FUNCTION_BLOCK FB_ITC_Conveyor IMPLEMENTS ITF_ITC
(**************************************************************************************
 *  Application     :   BoxControl Framework
 *  Revision date   :   $Date: 2021-04-08 12:45:11 +0200 (tor, 08 apr 2021) $
 *  Author          :   CDC
 *	Purpose			:	ITC - Message Manager.
 *						Represents the interface between the application and the 
 *						communication. Serves as abstract layer to ensure application
 *						independency.
 * ------------------------------------------------------------------------------------
 *  © Swisslog AG
 *  Swisslog is not liable for any usage of this source code that is not agreed 
 *  on between Swisslog and the other party. The mandatory legal liability remains 
 *  unaffected.
 * ------------------------------------------------------------------------------------
 *  Revision History: 
 *
 *  VERSION DATE         INITIALS     DESCRIPTION
 *  0.0     DD.MM.YYYY   (name)       (explain customized modifications)
 *
 **************************************************************************************)
VAR_INPUT
	Config			: ST_CFG_ITC_ManagerConv; // Config
END_VAR

VAR
	Init			: BOOL; // Initialized
	fbDebugMsg		: FB_DebugMsg; // Debug instance
	DebugMsg		: T_MAXSTRING; // Debug msg
	Idx				: INT; // Index for general usage 
	eMsgType		: E_ITC_MsgTypeConv; // Message type conveyor
	Position		: ST_PositionIdent;
	SDI				: ST_ITC_SDI; // SDI
	GVR				: ST_ITC_GVR; // GVR
	ISR				: ST_ITC_ISR; // ISR
	TTC				: ST_ITC_TTC; // TTC
	TDR				: ST_ITC_TDR; // TDR
	FCQ				: ST_ITC_FCQ; // FCQ
	FSR				: ST_ITC_FSR; // FSR
	FSR_Empty		: ST_ITC_FSR; // FSR empty
	SCR				: ST_ITC_SCR; // SCR
	SSR				: ST_ITC_SSR; // SSR
	SSR_Empty		: ST_ITC_SSR; // SSR empty
	GCR				: ST_ITC_GCR; // GCR
	GSR				: ST_ITC_GSR; // GSR
	GSR_Empty		: ST_ITC_GSR; // GSR empty
	ECR				: ST_ITC_ECR; // ECR
	ESR				: ST_ITC_ESR; // ESR
	ESR_Empty		: ST_ITC_ESR; // ESR empty
	FCR				: ST_ITC_FCR; // FCR
	MCR				: ST_ITC_MCR; // MCR
	MCR_Empty		: ST_ITC_MCR; // MCR empty
	SIR				: ST_ITC_SIR; // SIR
	TUR				: ST_ITC_TUR; // TUR
	GDR				: ST_ITC_GDR; // GDR
	GDR_Empty		: ST_ITC_GDR; // GDR empty
	DAR				: ST_ITC_DAR; // DAR
	DAR_Empty		: ST_ITC_DAR; // DAR empty
	Data			: ST_ITC_GeneralData; // General data
	RAC				: ST_ITC_RAC; // RAC
	RDR				: ST_ITC_RDR; // RDR
END_VAR

VAR PERSISTENT
	Settings			: ST_CFG_ITC_ManagerConv; // Active configuration
END_VAR

(**************************************************************************************************************
   Body never called!
***************************************************************************************************************)
;

{attribute 'object_name' := 'M_AddData'}
METHOD M_AddData : BOOL
(**************************************************************************************
 * 	Application		:	BoxControl Framework
 *	Revision		:	$Revision: 474929 $
 *	Revision date	:	$Date: 2021-04-08 12:45:11 +0200 (tor, 08 apr 2021) $
 *	Last changed by	:	$Author: b7gessa $
 *	URL				:	$URL: http://almscdc.swisslog.com/repo/SWPD/Development/BoxControlFramework/20_Release/tags/R1.12.0/01_Software/BCF/BCF/JumpStart/20_Product/10_BCF/11_Conv/11_Com/11_ITC/FB_ITC_Conveyor.TcPOU $
 *
 *	Purpose			:	Add data to the system
 *
 * ------------------------------------------------------------------------------------
 *	Copyright Swisslog [IP AG], Switzerland. All rights reserved.
 * 
 * ------------------------------------------------------------------------------------
 *	
 * 	Revision History: 
 *
 * 	VERSION			DATE			INITIALS			DESCRIPTION
 *	0.1				01.01.2001		swl					Example
 *
 **************************************************************************************)
VAR_INPUT
	meChannelSrc	: E_MFCS_Channel;
	mMsgType		: INT;
	mpData			: PVOID;
	mLen			: UDINT;
END_VAR

M_AddData := FALSE;
// Translate type to enumeration
eMsgType := mMsgType;

// Go to corresponding type
CASE eMsgType OF
	(****************************************************
	  No Message type
	*****************************************************)	
	E_ITC_MsgTypeConv.NO_MESSAGE_TYPE:
		;
	
	(****************************************************
	  Visualization information request
	*****************************************************)	
	E_ITC_MsgTypeConv.VISUALIZATION_INFORMATION_REQUEST:
		// Process
		M_AddData := M_ProcessVIQ(
						meChannelSrc := meChannelSrc,
						mpVIQ := mpData,
						mLen := mLen);
		
	(****************************************************
	  Digital input request
	*****************************************************)	
	E_ITC_MsgTypeConv.DIGITAL_INPUT_REQUEST:
		// Process
		M_AddData := M_ProcessDIQ(
						meChannelSrc := meChannelSrc);
		
	(****************************************************
	  Element control request
	*****************************************************)
	E_ITC_MsgTypeConv.ELEMENT_CONTROL_REQUEST:
		// Process
		M_AddData := M_ProcessECQ(
						meChannelSrc := meChannelSrc,
						mpECQ		 := mpData,
						mLen 		 := mLen);
	
	(****************************************************
	  Element status request
	*****************************************************)		
	E_ITC_MsgTypeConv.ELEMENT_STATUS_REQUEST:
		// Process
		M_AddData := M_ProcessESQ(
						meChannelSrc := meChannelSrc,
						mpESQ		 := mpData,
						mLen 	     := mLen);
		
	(****************************************************
	  Function control request
	*****************************************************)	
	E_ITC_MsgTypeConv.FUNCTION_CONTROL_REQUEST:
		// Process
		M_AddData := M_ProcessFCQ(
						meChannelSrc := meChannelSrc,
						mpFCQ		 := mpData,
						mLen 		 := mLen);
		
	(****************************************************
	  Function status request
	*****************************************************)	
	E_ITC_MsgTypeConv.FUNCTION_STATUS_REQUEST:
		// Process
		M_AddData := M_ProcessFSQ(
						meChannelSrc := meChannelSrc,
						mpFSQ		 := mpData,
						mLen 		 := mLen);
						
	(****************************************************
	  Group control request
	*****************************************************)				
	E_ITC_MsgTypeConv.GROUP_CONTROL_REQUEST:
		// Process
		M_AddData := M_ProcessGCQ(
						meChannelSrc := meChannelSrc,
						mpGCQ		 := mpData,
						mLen 		 := mLen);

	(****************************************************
	  Group status request
	*****************************************************)	
	E_ITC_MsgTypeConv.GROUP_STATUS_REQUEST:
		// Process
		M_AddData := M_ProcessGSQ(
						meChannelSrc := meChannelSrc,
						mpGSQ		 := mpData,
						mLen 		 := mLen);
		
	(****************************************************
	  Global variable request
	*****************************************************)	
	E_ITC_MsgTypeConv.GLOBAL_VARIABLE_REQUEST:
		// Process
		M_AddData := M_ProcessGVQ(
						meChannelSrc := meChannelSrc,
						mpGVQ := mpData,
						mLen := mLen);
						
	(****************************************************
	  IRQ request
	*****************************************************)	
	E_ITC_MsgTypeConv.I_O_STATUS_REQUEST:
		// Process
		M_AddData := M_ProcessIRQ(
						meChannelSrc := meChannelSrc,
						mpIRQ		 := mpData,
						mLen 	     := mLen);
		
	(****************************************************
	  Manual control request
	*****************************************************)					
	E_ITC_MsgTypeConv.MANUAL_CONTROL_REQUEST:
		// Process
		M_AddData := M_ProcessMCQ(
						meChannelSrc := meChannelSrc,
						mpMCQ		 := mpData,
						mLen 		 := mLen);
		
	(****************************************************
	  Robot action assignement
	*****************************************************)					
	E_ITC_MsgTypeConv.ROBOT_ACTION_ASSIGNMENT:
		// Process
		M_AddData := M_ProcessRAA(
						meChannelSrc := meChannelSrc,
						mpRAA		 := mpData,
						mLen 		 := mLen);		
				
	(****************************************************
	  Robot delete request
	*****************************************************)					
	E_ITC_MsgTypeConv.ROBOT_DELETE_REQUEST:
		// Process
		M_AddData := M_ProcessRDQ(
						meChannelSrc := meChannelSrc,
						mpRDQ		 := mpData,
						mLen 		 := mLen);	
			
	(****************************************************
	  Subsystem control request
	*****************************************************)				
	E_ITC_MsgTypeConv.SUBSYSTEM_CONTROL_REQUEST:
		// Process
		M_AddData := M_ProcessSCQ(
						meChannelSrc := meChannelSrc,
						mpSCQ		 := mpData,
						mLen 		 := mLen);
		
	(****************************************************
	  Set digital output
	*****************************************************)				
	E_ITC_MsgTypeConv.SET_DIGITAL_OUTPUT:
		// Process
		M_AddData := M_ProcessSDO(
						meChannelSrc := meChannelSrc,
						mpSDO		 := mpData,
						mLen 		 := mLen);
		
	(****************************************************
	  Scanner information request
	*****************************************************)				
	E_ITC_MsgTypeConv.SCANNER_INFORMATION_REQUEST:
		// Process
		M_AddData := M_ProcessSIQ(
						meChannelSrc := meChannelSrc,
						mpSIQ		 := mpData,
						mLen 		 := mLen);
		
	(****************************************************
	  Subsystem status request
	*****************************************************)			
	E_ITC_MsgTypeConv.SUBSYSTEM_STATUS_REQUEST:
		// Process
		M_AddData := M_ProcessSSQ(
						meChannelSrc := meChannelSrc,
						mpSSQ		 := mpData,
						mLen 		 := mLen);
		
	(****************************************************
	  Task delete request
	*****************************************************)			
	E_ITC_MsgTypeConv.TASK_DELETE_REQUEST:
		// Process
		M_AddData := M_ProcessTDQ(
						meChannelSrc := meChannelSrc,
						mpTDQ		 := mpData,
						mLen 		 := mLen);
		
	(****************************************************
	  Transport task assignment
	*****************************************************)	
	E_ITC_MsgTypeConv.TRANSPORT_TASK_ASSIGNMENT:
		// Process
		M_AddData := M_ProcessTTA(
						meChannelSrc := meChannelSrc,
						mpTTA		 := mpData,
						mLen 		 := mLen);
		
	(****************************************************
	  Transport unit request
	*****************************************************)	
	E_ITC_MsgTypeConv.TRANSPORT_UNIT_REQUEST:
		// Process
		M_AddData := M_ProcessTUQ(
						meChannelSrc := meChannelSrc,
						mpTUQ		 := mpData,
						mLen 	     := mLen);

	(****************************************************
	  Add TU data index into function
	*****************************************************)	
	E_ITC_MsgTypeConv.ADD_TU_DATA:
		// Process
		M_AddData := M_AddTUData(
						meChannelSrc := meChannelSrc,
						mpAddTU_Data		 := mpData);					


						
	(****************************************************
		Data Aquisition Request 
	*****************************************************)	
	E_ITC_MsgTypeConv.DATA_ACQUISITION_REQUEST:
		// Process
		M_AddData := M_ProcessDAQ(
						meChannelSrc := meChannelSrc,
						mpDAQ		 := mpData,
						mLen 	     := mLen);
	(****************************************************
		Gathered Data  Request 
	*****************************************************)	
	E_ITC_MsgTypeConv.GATHERED_DATA_REQUEST:
		// Process
		M_AddData := M_ProcessGDQ(
						meChannelSrc := meChannelSrc,
						mpGDQ		 := mpData,
						mLen 	     := mLen);				
ELSE
	// Unknown type
	DebugMsg := 'Unknown message type received';
	fbDebugMsg.M_SendErrorMsg(mMessage := DebugMsg);		
END_CASE
END_METHOD

METHOD PROTECTED M_AddTUData : BOOL

(**************************************************************************************
 * 	Application		:	BoxControl Framework
 *	Revision		:	$Revision: 474929 $
 *	Revision date	:	$Date: 2021-04-08 12:45:11 +0200 (tor, 08 apr 2021) $
 *	Last changed by	:	$Author: b7gessa $
 *	URL				:	$URL: http://almscdc.swisslog.com/repo/SWPD/Development/BoxControlFramework/20_Release/tags/R1.12.0/01_Software/BCF/BCF/JumpStart/20_Product/10_BCF/11_Conv/11_Com/11_ITC/FB_ITC_Conveyor.TcPOU $
 *
 *	Purpose			:	Process a received Digital Input Request telegram.
 *
 * ------------------------------------------------------------------------------------
 *	Copyright Swisslog [IP AG], Switzerland. All rights reserved.
 * 
 * ------------------------------------------------------------------------------------
 *	
 * 	Revision History: 
 *
 * 	VERSION			DATE			INITIALS			DESCRIPTION
 *	0.1				01.01.2001		swl					Example
 *
 **************************************************************************************)
VAR_INPUT
	meChannelSrc		: E_MFCS_Channel; // Source communicaton channel
	mpAddTU_Data		: POINTER TO ST_ITC_ADD_TU_DATA; // Pointer to SCQ
END_VAR
Data.Init := TRUE;
Data.TU_DataIndex := mpAddTU_Data^.TU_DataIndex;
Data.ZoneNumber := mpAddTU_Data^.ZoneNumber;
Data.Position := '';

// Forward to position
M_AddTUData := M_ProcessToFunction(
	meFunctionNumber	:= mpAddTU_Data^.eFunctionNumber, 
	meChannelSrc		:= meChannelSrc, 
	mMsgType			:= E_ITC_MsgTypeConv.ADD_TU_DATA,
	mpData				:= ADR(Data), 
	mLen				:= SIZEOF(Data));
END_METHOD

{attribute 'object_name' := 'M_CallITC_Service'}
METHOD M_CallITC_Service : BOOL
VAR
	mIdx : INT;
END_VAR
(**************************************************************************************************************
 	Initialization
***************************************************************************************************************)
M_Init(FALSE);

(**************************************************************************************************************
  Monitor SDI Signals
***************************************************************************************************************)
FOR mIdx := 1 TO Settings.SDI_Limit DO
	// SDI signal is enabled 
	IF SDISignalNumber[mIdx].Enabled THEN
		// SDI signal changed state 
		IF SDISignalNumber[mIdx].State <> SDISignalNumber[mIdx].LastState THEN
			// Send SDI
			F_ITC_SendSDI(
				eChannelSrc		:= 0, 
				SignalNumber	:= mIdx, 
				SignalState		:= SDISignalNumber[mIdx].State, 
				eReturnCode		:= E_ErrorConv.NO_ERROR_CODE);
				
			// Update state
			SDISignalNumber[mIdx].LastState := SDISignalNumber[mIdx].State;
		END_IF
	END_IF
END_FOR
END_METHOD

METHOD M_Init : BOOL
(**************************************************************************************
 * 	Application		:	BoxControl Framework
 *	Revision		:	$Revision: 474929 $
 *	Revision date	:	$Date: 2021-04-08 12:45:11 +0200 (tor, 08 apr 2021) $
 *	Last changed by	:	$Author: b7gessa $
 *	URL				:	$URL: http://almscdc.swisslog.com/repo/SWPD/Development/BoxControlFramework/20_Release/tags/R1.12.0/01_Software/BCF/BCF/JumpStart/20_Product/10_BCF/11_Conv/11_Com/11_ITC/FB_ITC_Conveyor.TcPOU $
 *
 *	Purpose			:	Initialize.
 *
 * ------------------------------------------------------------------------------------
 *	Copyright Swisslog [IP AG], Switzerland. All rights reserved.
 * 
 * ------------------------------------------------------------------------------------
 *	
 * 	Revision History: 
 *
 * 	VERSION			DATE			INITIALS			DESCRIPTION
 *	0.1				01.01.2001		swl					Example
 *
 **************************************************************************************)
VAR_INPUT
	mInit		: BOOL; // Force init
END_VAR
// If instance is not initialized or init is forced
IF mInit OR NOT Init THEN
	// Update configuration
	Settings := Config;
	
	// Send log message
    fbDebugMsg.M_SendInfoMsg('Initialization done');
		
	// Init done
    Init := TRUE;
END_IF
END_METHOD

METHOD PRIVATE M_ProcessDAQ : BOOL
(**************************************************************************************
 * 	Application		:	BoxControl Framework
 *	Revision		:	$Revision: 474929 $
 *	Revision date	:	$Date: 2021-04-08 12:45:11 +0200 (tor, 08 apr 2021) $
 *	Last changed by	:	$Author: b7gessa $
 *	URL				:	$URL: http://almscdc.swisslog.com/repo/SWPD/Development/BoxControlFramework/20_Release/tags/R1.12.0/01_Software/BCF/BCF/JumpStart/20_Product/10_BCF/11_Conv/11_Com/11_ITC/FB_ITC_Conveyor.TcPOU $
 *
 *	Purpose			:	Process a received Data Aquisition telegram.
 *
 * ------------------------------------------------------------------------------------
 *	Copyright Swisslog [IP AG], Switzerland. All rights reserved.
 * 
 * ------------------------------------------------------------------------------------
 *	
 * 	Revision History: 
 *
 * 	VERSION			DATE			INITIALS			DESCRIPTION
 *	0.1				01.01.2001		swl					Example
 *
 **************************************************************************************)
VAR_INPUT
	meChannelSrc		: E_MFCS_Channel; // Source communicaton channel
	mpDAQ				: POINTER TO ST_ITC_DAQ; // Pointer to DAQ
	mLen				: UDINT; // Data length
END_VAR
VAR
	meFunctionPosition		: ST_PositionIdent; // Position
	meGroupNumber			: E_GroupNumber; // Group
	meElementNumber			: E_ElementNumber;//Element Number
	meSubsystem				: BOOL;	//Subsystem
	mReturnCode				: E_ErrorConv; // Error code

END_VAR
// Initialize
M_ProcessDAQ:= TRUE;

//Check where position is
meFunctionPosition := F_SearchFunctionPosition(Position := mpDAQ^.Position);
meElementNumber    := F_SearchElementPosition(ElementName := mpDAQ^.Position);
meGroupNumber      := F_SearchGroupNumber(GroupName := mpDAQ^.Position);
meSubsystem 	   := F_EqualSisNames(Name1 := SubsystemRegistry.SubSystemName,
									Name2 := mpDAQ^.Position);

// Check if Function Number is valid
IF meFunctionPosition.eFunctionNumber >F_BEGIN_FUNCTION AND
	meFunctionPosition.eFunctionNumber <F_END_FUNCTION THEN 
    // Forward to Function
	M_ProcessDAQ := M_ProcessToFunction(
						meFunctionNumber:= 	meFunctionPosition.eFunctionNumber, // Position
						meChannelSrc	:= meChannelSrc, 
						mpData			:= mpDAQ, 
						mMsgType		:= E_ITC_MsgTypeConv.DATA_ACQUISITION_REQUEST,
						mLen			:= mLen);
// Check if DAQ was sent to an Element	
ELSIF meElementNumber > E_ElementNumber.E_BEGIN_ELEMENT AND 
      meElementNumber < E_ElementNumber.E_END_ELEMENT AND
      meFunctionPosition.eFunctionNumber = F_BEGIN_FUNCTION AND
      meFunctionPosition.ZoneNumber = 0 THEN 
		// Forward to element
		M_ProcessDAQ := M_ProcessToElement(
						meElementNumber	:= meElementNumber, 
						meChannelSrc	:= meChannelSrc, 
						mpData			:= mpDAQ, 
						mMsgType		:= E_ITC_MsgTypeConv.DATA_ACQUISITION_REQUEST,
						mLen			:= mLen);
// Check if DAQ was sent to a Group					
ELSIF  meGroupNumber > E_GroupNumber.G_BEGIN_GROUP AND 
   		meGroupNumber < E_GroupNumber.G_END_GROUP   AND
		meElementNumber 					= E_BEGIN_ELEMENT AND 
      	meFunctionPosition.eFunctionNumber 	= F_BEGIN_FUNCTION AND
      	meFunctionPosition.ZoneNumber 		= 0 THEN 	   
		// Forward to Group
		M_ProcessDAQ := M_ProcessToGroup(
							meGroupNumber	:= meGroupNumber, // Groupnumber
							meChannelSrc	:= meChannelSrc, 
							mpData			:= mpDAQ, 
							mMsgType		:= E_ITC_MsgTypeConv.DATA_ACQUISITION_REQUEST,
							mLen			:= mLen);
// Check if DAQ was sent to a SubSystem
ELSIF  meSubsystem AND
	   meGroupNumber = G_BEGIN_GROUP AND
	   meElementNumber = E_BEGIN_ELEMENT AND 
	   meFunctionPosition.eFunctionNumber = F_BEGIN_FUNCTION AND
	   meFunctionPosition.ZoneNumber = 0 THEN 	   		
	// Forward to Subsytem						
	M_ProcessDAQ := M_ProcessToSubsystem(
						meChannelSrc	:= meChannelSrc, 
						mpData			:= mpDAQ, 
						mMsgType		:= E_ITC_MsgTypeConv.DATA_ACQUISITION_REQUEST,
						mLen			:= mLen);					
ELSE
	//Unknown position send DAR with Error Report	
	DAR := DAR_Empty;
	// DAR
	DAR.Position	:= mpDAQ^.Position;
	DAR.eErrorCode	:= E_ErrorConv.ELEMENTNUMBER_UNKNOWN;

	// Reject telegram	
	M_SendData(
		meChannel := meChannelSrc,
		mMsgType  := E_ITC_MsgTypeConv.DATA_ACQUISITION_REPORT,
		mpData    := ADR(DAR),
		mLen	  := SIZEOF(DAR));
		
	// Unknown Position name received
	DebugMsg := CONCAT('DAQ - unknown Position name received: ', mpDAQ^.Position);
	fbDebugMsg.M_SendErrorMsg(mMessage := DebugMsg);
END_IF
END_METHOD

METHOD PROTECTED M_ProcessDIQ : BOOL
(**************************************************************************************
 * 	Application		:	BoxControl Framework
 *	Revision		:	$Revision: 474929 $
 *	Revision date	:	$Date: 2021-04-08 12:45:11 +0200 (tor, 08 apr 2021) $
 *	Last changed by	:	$Author: b7gessa $
 *	URL				:	$URL: http://almscdc.swisslog.com/repo/SWPD/Development/BoxControlFramework/20_Release/tags/R1.12.0/01_Software/BCF/BCF/JumpStart/20_Product/10_BCF/11_Conv/11_Com/11_ITC/FB_ITC_Conveyor.TcPOU $
 *
 *	Purpose			:	Process a received Digital Input Request telegram.
 *
 * ------------------------------------------------------------------------------------
 *	Copyright Swisslog [IP AG], Switzerland. All rights reserved.
 * 
 * ------------------------------------------------------------------------------------
 *	
 * 	Revision History: 
 *
 * 	VERSION			DATE			INITIALS			DESCRIPTION
 *	0.1				01.01.2001		swl					Example
 *
 **************************************************************************************)
VAR_INPUT
	meChannelSrc			: E_MFCS_Channel; // Source communicaton channel
END_VAR
// Compose an SDI telegram for every enabled SDI signal
FOR Idx := 1 TO NUMBER_OF_SDI_SIGNALS DO
	// For all enabled SDI SignalNumbers
	IF SDISignalNumber[Idx].Enabled THEN
		// Collect data
		SDI.SignalNumber := Idx;
		SDI.SignalState  := SDISignalNumber[Idx].State;
		SDI.ReturnCode	 := E_ErrorConv.NO_ERROR_CODE;
	
		M_SendData(
			meChannel := meChannelSrc, 
			mMsgType  := E_ITC_MsgTypeConv.SEND_DIGITAL_INPUT, 
			mpData    := ADR(SDI),
			mLen	  := SIZEOF(SDI));
	END_IF
END_FOR

// Telegram processed
M_ProcessDIQ := TRUE;
END_METHOD

METHOD PROTECTED M_ProcessECQ : BOOL
(**************************************************************************************
 * 	Application		:	BoxControl Framework
 *	Revision		:	$Revision: 474929 $
 *	Revision date	:	$Date: 2021-04-08 12:45:11 +0200 (tor, 08 apr 2021) $
 *	Last changed by	:	$Author: b7gessa $
 *	URL				:	$URL: http://almscdc.swisslog.com/repo/SWPD/Development/BoxControlFramework/20_Release/tags/R1.12.0/01_Software/BCF/BCF/JumpStart/20_Product/10_BCF/11_Conv/11_Com/11_ITC/FB_ITC_Conveyor.TcPOU $
 *
 *	Purpose			:	Process a received Element Control Request 
 *
 * ------------------------------------------------------------------------------------
 *	Copyright Swisslog [IP AG], Switzerland. All rights reserved.
 * 
 * ------------------------------------------------------------------------------------
 *	
 * 	Revision History: 
 *
 * 	VERSION			DATE			INITIALS			DESCRIPTION
 *	0.1				01.01.2001		swl					Example
 *
 **************************************************************************************)
VAR_INPUT
	meChannelSrc		: E_MFCS_Channel; // Source communicaton channel
	mpECQ				: POINTER TO ST_ITC_ECQ; // Pointer to ECQ
	mLen				: UDINT; // Data length
END_VAR

VAR
	meElementNumber		: E_ElementNumber; // Element number
END_VAR
// Initialize
M_ProcessECQ := TRUE;

// Try getting enum
meElementNumber := F_SearchElementPosition(ElementName := mpECQ^.Position);

// Check if ElementNumber is valid
IF meElementNumber > E_ElementNumber.E_BEGIN_ELEMENT AND 
   meElementNumber < E_ElementNumber.E_END_ELEMENT THEN
			
	// Forward to element
	M_ProcessECQ := M_ProcessToElement(
						meElementNumber	:= meElementNumber, 
						meChannelSrc	:= meChannelSrc, 
						mMsgType		:= E_ITC_MsgTypeConv.ELEMENT_CONTROL_REQUEST,
						mpData			:= mpECQ, 
						mLen			:= mLen);
						
ELSE
	// Unknown Position name received
	// ECR
	ECR.Position	:= mpECQ^.Position;
	ECR.Code		:= mpECQ^.Code;
	ECR.Variable	:= mpECQ^.Variable;
	ECR.ReturnCode	:= E_ErrorConv.ELEMENTNUMBER_UNKNOWN;

	// Reject telegram	
	M_SendData(
		meChannel := meChannelSrc,
		mMsgType  := E_ITC_MsgTypeConv.ELEMENT_CONTROL_REPLY,
		mpData    := ADR(ECR),
		mLen	  := SIZEOF(ECR));
		
	// Unknown Position name received
	DebugMsg := CONCAT('ECQ - unknown Position name received: ', mpECQ^.Position);
	fbDebugMsg.M_SendErrorMsg(mMessage := DebugMsg);
END_IF
END_METHOD

METHOD PROTECTED M_ProcessESQ : BOOL
(**************************************************************************************
 * 	Application		:	BoxControl Framework
 *	Revision		:	$Revision: 474929 $
 *	Revision date	:	$Date: 2021-04-08 12:45:11 +0200 (tor, 08 apr 2021) $
 *	Last changed by	:	$Author: b7gessa $
 *	URL				:	$URL: http://almscdc.swisslog.com/repo/SWPD/Development/BoxControlFramework/20_Release/tags/R1.12.0/01_Software/BCF/BCF/JumpStart/20_Product/10_BCF/11_Conv/11_Com/11_ITC/FB_ITC_Conveyor.TcPOU $
 *
 *	Purpose			:	Process a received Element Status Request telegram.
 *
 * ------------------------------------------------------------------------------------
 *	Copyright Swisslog [IP AG], Switzerland. All rights reserved.
 * 
 * ------------------------------------------------------------------------------------
 *	
 * 	Revision History: 
 *
 * 	VERSION			DATE			INITIALS			DESCRIPTION
 *	0.1				01.01.2001		swl					Example
 *
 **************************************************************************************)
VAR_INPUT
	meChannelSrc		: E_MFCS_Channel; // Source communicaton channel
	mpESQ				: POINTER TO ST_ITC_ESQ; // Pointer to ESQ
	mLen				: UDINT; // Data length
END_VAR

VAR
	meElementNumber		: E_ElementNumber; // Element number
END_VAR
// Initialize
M_ProcessESQ := TRUE;

// Try getting enum
meElementNumber := F_SearchElementPosition(ElementName := mpESQ^.Position);

// Check if ElementNumber is valid
IF meElementNumber > E_ElementNumber.E_BEGIN_ELEMENT AND 
   meElementNumber < E_ElementNumber.E_END_ELEMENT THEN			
	
	// Forward to element
	M_ProcessESQ := M_ProcessToElement(
						meElementNumber	:= meElementNumber, 
						meChannelSrc	:= meChannelSrc, 
						mMsgType		:= E_ITC_MsgTypeConv.ELEMENT_STATUS_REQUEST,
						mpData			:= mpESQ, 
						mLen			:= mLen);
						
// Check if ESQ was sent to a SubSystem
ELSIF F_EqualSisNames(Name1 := SubsystemRegistry.SubSystemName,
                      Name2 := mpESQ^.Position) THEN
									
	// Do for each ElementNumber
	FOR meElementNumber := E_ElementNumber.E_BEGIN_ELEMENT + 1 TO E_ElementNumber.E_END_Element - 1 DO
		// Forward
		M_ProcessToElement(
			meElementNumber	:= meElementNumber, 
			meChannelSrc	:= meChannelSrc, 
			mMsgType		:= E_ITC_MsgTypeConv.ELEMENT_STATUS_REQUEST,
			mpData			:= mpESQ, 
			mLen			:= mLen);
	END_FOR
ELSE
	ESR := ESR_Empty;
	// Unknown Position name received
	// ESR
	ESR.Position	:= mpESQ^.Position;
	ESR.ReturnCode	:= E_ErrorConv.ELEMENTNUMBER_UNKNOWN;

	// Reject telegram	
	M_SendData(
		meChannel := meChannelSrc,
		mMsgType  := E_ITC_MsgTypeConv.ELEMENT_STATUS_REPORT,
		mpData    := ADR(ESR),
		mLen	  := SIZEOF(ESR));
		
	// Unknown Position name received
	DebugMsg := CONCAT('ESQ - unknown Position name received: ', mpESQ^.Position);
	fbDebugMsg.M_SendErrorMsg(mMessage := DebugMsg);
END_IF
END_METHOD

METHOD PROTECTED M_ProcessFCQ : BOOL
(**************************************************************************************
 * 	Application		:	BoxControl Framework
 *	Revision		:	$Revision: 474929 $
 *	Revision date	:	$Date: 2021-04-08 12:45:11 +0200 (tor, 08 apr 2021) $
 *	Last changed by	:	$Author: b7gessa $
 *	URL				:	$URL: http://almscdc.swisslog.com/repo/SWPD/Development/BoxControlFramework/20_Release/tags/R1.12.0/01_Software/BCF/BCF/JumpStart/20_Product/10_BCF/11_Conv/11_Com/11_ITC/FB_ITC_Conveyor.TcPOU $
 *
 *	Purpose			:	Process a received Function Control Request.
 *
 * ------------------------------------------------------------------------------------
 *	Copyright Swisslog [IP AG], Switzerland. All rights reserved.
 * 
 * ------------------------------------------------------------------------------------
 *	
 * 	Revision History: 
 *
 * 	VERSION			DATE			INITIALS			DESCRIPTION
 *	0.1				01.01.2001		swl					Example
 *
 **************************************************************************************)
VAR_INPUT
	meChannelSrc		: E_MFCS_Channel; // Source communicaton channel
	mpFCQ				: POINTER TO ST_ITC_FCQ; // Pointer to FCQ
	mLen				: UDINT; // Data length
END_VAR

VAR
	mMsgPosition		: ST_PositionIdent; // Function position
	mrefObject			: REFERENCE TO FB_BaseObject; // Reference
END_VAR
// Initialize
M_ProcessFCQ := TRUE;

// Get position from message
mMsgPosition := F_SearchFunctionPosition(Position := mpFCQ^.Position);

// If a valid function was found with a valid zone
IF 	mMsgPosition.eFunctionNumber > E_FunctionNumber.F_BEGIN_FUNCTION AND 
	mMsgPosition.eFunctionNumber < E_FunctionNumber.F_END_FUNCTION AND 
	mMsgPosition.ZoneNumber >= 0 AND mMsgPosition.ZoneNumber <= NUMBER_OF_ZONES_PER_FUNCTION THEN
	
	// Forward to element
	M_ProcessFCQ := M_ProcessToFunction(
						meFunctionNumber	:= mMsgPosition.eFunctionNumber, 
						meChannelSrc		:= meChannelSrc, 
						mMsgType			:= E_ITC_MsgTypeConv.FUNCTION_CONTROL_REQUEST,
						mpData				:= mpFCQ, 
						mLen				:= mLen);
						
ELSE
	// FCR
	FCR.Position	:= mpFCQ^.Position;
	FCR.Code		:= mpFCQ^.Code;
	FCR.Variable	:= mpFCQ^.Variable;
	FCR.ReturnCode	:= E_ErrorConv.FUNCTIONNUMBER_UNKNOWN;

	// Reject telegram	
	M_SendData(
		meChannel := meChannelSrc,
		mMsgType  := E_ITC_MsgTypeConv.FUNCTION_CONTROL_REPLY,
		mpData    := ADR(FCR),
        mLen	  := SIZEOF(FCR));
		
	// Unknown Position name received 
	DebugMsg := CONCAT('FCQ, Unknown Position received: ', mpFCQ^.Position);
	fbDebugMsg.M_SendErrorMsg(mMessage := DebugMsg); 
END_IF
END_METHOD

METHOD PROTECTED M_ProcessFSQ : BOOL
(**************************************************************************************
 * 	Application		:	BoxControl Framework
 *	Revision		:	$Revision: 474929 $
 *	Revision date	:	$Date: 2021-04-08 12:45:11 +0200 (tor, 08 apr 2021) $
 *	Last changed by	:	$Author: b7gessa $
 *	URL				:	$URL: http://almscdc.swisslog.com/repo/SWPD/Development/BoxControlFramework/20_Release/tags/R1.12.0/01_Software/BCF/BCF/JumpStart/20_Product/10_BCF/11_Conv/11_Com/11_ITC/FB_ITC_Conveyor.TcPOU $
 *
 *	Purpose			:	Process a received position Status Request telegram.
 *
 * ------------------------------------------------------------------------------------
 *	Copyright Swisslog [IP AG], Switzerland. All rights reserved.
 * 
 * ------------------------------------------------------------------------------------
 *	
 * 	Revision History: 
 *
 * 	VERSION			DATE			INITIALS			DESCRIPTION
 *	0.1				01.01.2001		swl					Example
 *
 **************************************************************************************)
VAR_INPUT
	meChannelSrc		: E_MFCS_Channel; // Source communicaton channel
	mpFSQ				: POINTER TO ST_ITC_FSQ; // Pointer to FSQ
	mLen				: UDINT; // Data length
END_VAR

VAR
	mMsgPosition		: ST_PositionIdent; // Function position
	mrefObject			: REFERENCE TO FB_BaseObject; // Reference
END_VAR
// Initialize
M_ProcessFSQ := TRUE;

// Get position from message
mMsgPosition := F_SearchFunctionPosition(Position := mpFSQ^.Position);

// If a valid function was found with a valid zone
IF 	mMsgPosition.eFunctionNumber > E_FunctionNumber.F_BEGIN_FUNCTION AND 
	mMsgPosition.eFunctionNumber < E_FunctionNumber.F_END_FUNCTION AND 
	mMsgPosition.ZoneNumber >= 0 AND mMsgPosition.ZoneNumber <= NUMBER_OF_ZONES_PER_FUNCTION THEN

	// Forward to element
	M_ProcessFSQ := M_ProcessToFunction(
						meFunctionNumber	:= mMsgPosition.eFunctionNumber, 
						meChannelSrc		:= meChannelSrc, 
						mMsgType			:= E_ITC_MsgTypeConv.FUNCTION_STATUS_REQUEST,
						mpData				:= mpFSQ,
						mLen				:= mLen);

ELSE
	
	FSR := FSR_Empty;
	
	// FSR
	FSR.Position	:= mpFSQ^.Position;
	FSR.eReturnCode	:= E_ErrorConv.FUNCTIONNUMBER_UNKNOWN;

	// Reject telegram	
	M_SendData(
		meChannel := meChannelSrc,
		mMsgType  := E_ITC_MsgTypeConv.FUNCTION_STATUS_REPORT,
		mpData    := ADR(FSR),
		mLen	  := SIZEOF(FSR));
		
	// Unknown Position name received 
	DebugMsg := CONCAT('FSQ, Unknown Position received: ', mpFSQ^.Position);
	fbDebugMsg.M_SendErrorMsg(mMessage := DebugMsg); 
END_IF
END_METHOD

METHOD PROTECTED M_ProcessGCQ : BOOL
(**************************************************************************************
 * 	Application		:	BoxControl Framework
 *	Revision		:	$Revision: 474929 $
 *	Revision date	:	$Date: 2021-04-08 12:45:11 +0200 (tor, 08 apr 2021) $
 *	Last changed by	:	$Author: b7gessa $
 *	URL				:	$URL: http://almscdc.swisslog.com/repo/SWPD/Development/BoxControlFramework/20_Release/tags/R1.12.0/01_Software/BCF/BCF/JumpStart/20_Product/10_BCF/11_Conv/11_Com/11_ITC/FB_ITC_Conveyor.TcPOU $
 *
 *	Purpose			:	Process a received Group Control Request telegram.
 *
 * ------------------------------------------------------------------------------------
 *	Copyright Swisslog [IP AG], Switzerland. All rights reserved.
 * 
 * ------------------------------------------------------------------------------------
 *	
 * 	Revision History: 
 *
 * 	VERSION			DATE			INITIALS			DESCRIPTION
 *	0.1				01.01.2001		swl					Example
 *
 **************************************************************************************)
VAR_INPUT
	meChannelSrc		: E_MFCS_Channel; // Source communicaton channel
	mpGCQ				: POINTER TO ST_ITC_GCQ; // Pointer to GCQ
	mLen				: UDINT; // Data length
END_VAR

VAR
	meGroupNumber		: E_GroupNumber; // group number
END_VAR
// Initialize 
M_ProcessGCQ := TRUE;

// Find GropuNumber of telegram
meGroupNumber := F_SearchGroupNumber(GroupName := mpGCQ^.Position);
			
// Group number valid
IF meGroupNumber > E_GroupNumber.G_BEGIN_GROUP AND 
   meGroupNumber < E_GroupNumber.G_END_GROUP THEN	
				
	// Forward to group
	M_ProcessGCQ := M_ProcessToGroup(
						meGroupNumber	:= meGroupNumber, 
						meChannelSrc	:= meChannelSrc, 
						mMsgType		:= E_ITC_MsgTypeConv.GROUP_CONTROL_REQUEST,
						mpData			:= mpGCQ, 
						mLen			:= mLen);
				
// Check if GCQ was sent to a SubSystem
ELSIF F_EqualSisNames(Name1 := SubsystemRegistry.SubSystemName,
                      Name2 := mpGCQ^.Position) THEN
			
	// Do for each GroupNumber
	FOR meGroupNumber := E_GroupNumber.G_BEGIN_GROUP + 1 TO E_GroupNumber.G_END_GROUP - 1 DO
		// Check if group is a switching group
		IF GroupRegistry[meGroupNumber].eGroupType = E_GroupType.SG THEN
			M_ProcessToGroup(
				meGroupNumber	:= meGroupNumber, 
				meChannelSrc	:= meChannelSrc, 
				mMsgType		:= E_ITC_MsgTypeConv.GROUP_CONTROL_REQUEST,
				mpData			:= mpGCQ, 
				mLen 			:= mLen);
		END_IF
	END_FOR
ELSE
	
	// GCR
	GCR.GroupName	:= mpGCQ^.Position;
	GCR.Code		:= mpGCQ^.Code;
	GCR.Variable	:= mpGCQ^.Variable;
	GCR.ReturnCode	:= E_ErrorConv.GROUPNUMBER_UNKNOWN;

	// Reject telegram	
	M_SendData(
		meChannel := meChannelSrc,
		mMsgType  := E_ITC_MsgTypeConv.GROUP_CONTROL_REPLY,
		mpData    := ADR(GCR),
		mLen	  := SIZEOF(GCR));

	// Unknown Group name received
	DebugMsg := CONCAT('GCQ, unknown Group name received: ', mpGCQ^.Position);
	fbDebugMsg.M_SendErrorMsg(mMessage := DebugMsg);
END_IF
END_METHOD

METHOD PROTECTED M_ProcessGDQ : BOOL
(**************************************************************************************
 * 	Application		:	BoxControl Framework
 *	Revision		:	$Revision: 474929 $
 *	Revision date	:	$Date: 2021-04-08 12:45:11 +0200 (tor, 08 apr 2021) $
 *	Last changed by	:	$Author: b7gessa $
 *	URL				:	$URL: http://almscdc.swisslog.com/repo/SWPD/Development/BoxControlFramework/20_Release/tags/R1.12.0/01_Software/BCF/BCF/JumpStart/20_Product/10_BCF/11_Conv/11_Com/11_ITC/FB_ITC_Conveyor.TcPOU $
 *
 *	Purpose			:	Process a received Gathered Data Request telegram.
 *
 * ------------------------------------------------------------------------------------
 *	Copyright Swisslog [IP AG], Switzerland. All rights reserved.
 * 
 * ------------------------------------------------------------------------------------
 *	
 * 	Revision History: 
 *
 * 	VERSION			DATE			INITIALS			DESCRIPTION
 *	0.1				01.01.2001		swl					Example
 *
 **************************************************************************************)
VAR_INPUT
	meChannelSrc		: E_MFCS_Channel; // Source communicaton channel
	mpGDQ				: POINTER TO ST_ITC_GDQ; // Pointer to GDQ
	mLen				: UDINT; // Data length
END_VAR
VAR
	meFunctionPosition				: ST_PositionIdent; // Position
	meGroupNumber					: E_GroupNumber; // Group
	meElementNumber					: E_ElementNumber;//Element Number
	meSubsystem						: BOOL;	
	mReturnCode						: E_ErrorConv; // Error code
END_VAR
// Initialize
M_ProcessGDQ:= TRUE;

//Search Position
meFunctionPosition := F_SearchFunctionPosition(Position := mpGDQ^.Position);
meElementNumber    := F_SearchElementPosition(ElementName := mpGDQ^.Position);
meGroupNumber      := F_SearchGroupNumber(GroupName := mpGDQ^.Position);
meSubsystem 	   := F_EqualSisNames(Name1 := SubsystemRegistry.SubSystemName,
														        Name2 := mpGDQ^.Position);

// Check if Function is Target for Telgram 
IF meFunctionPosition.eFunctionNumber >F_BEGIN_FUNCTION AND
	meFunctionPosition.eFunctionNumber <F_END_FUNCTION THEN 
    // Forward to Function
	M_ProcessGDQ := M_ProcessToFunction(
						meFunctionNumber:= 	meFunctionPosition.eFunctionNumber, // Position
						meChannelSrc	:= meChannelSrc, 
						mpData			:= mpGDQ, 
						mMsgType		:= E_ITC_MsgTypeConv.GATHERED_DATA_REQUEST,
						mLen			:= mLen);
// Check if Element is Target for Telgram 
ELSIF meElementNumber > E_ElementNumber.E_BEGIN_ELEMENT AND 
      meElementNumber < E_ElementNumber.E_END_ELEMENT AND
      meFunctionPosition.eFunctionNumber = F_BEGIN_FUNCTION AND
      meFunctionPosition.ZoneNumber = 0 THEN 
	// Forward to element
	M_ProcessGDQ := M_ProcessToElement(
						meElementNumber	:= meElementNumber, 
						meChannelSrc	:= meChannelSrc, 
						mpData			:= mpGDQ, 
						mMsgType		:= E_ITC_MsgTypeConv.GATHERED_DATA_REQUEST,
						mLen			:= mLen);

// Check if Group is Target for Telgram 				
ELSIF  	meGroupNumber > E_GroupNumber.G_BEGIN_GROUP AND 
   		meGroupNumber < E_GroupNumber.G_END_GROUP   AND
		meElementNumber 					= E_BEGIN_ELEMENT AND 
      	meFunctionPosition.eFunctionNumber 	= F_BEGIN_FUNCTION AND
      	meFunctionPosition.ZoneNumber 		= 0 THEN 	   
			
		// Forward to Group
		M_ProcessGDQ := M_ProcessToGroup(
											meGroupNumber	:= meGroupNumber, // Groupnumber
											meChannelSrc	:= meChannelSrc, 
											mpData			:= mpGDQ, 
											mMsgType		:= E_ITC_MsgTypeConv.GATHERED_DATA_REQUEST,
											mLen			:= mLen);
	 
		
// Check if Subystem Target for Telgram 
ELSIF  meSubsystem AND
	   meGroupNumber = G_BEGIN_GROUP AND
	   meElementNumber = E_BEGIN_ELEMENT AND 
	   meFunctionPosition.eFunctionNumber = F_BEGIN_FUNCTION AND
	   meFunctionPosition.ZoneNumber = 0 THEN 	   	
		// Forward to Subsytem			
		M_ProcessGDQ := M_ProcessToSubsystem(
							meChannelSrc	:= meChannelSrc, 
							mpData			:= mpGDQ, 
							mMsgType		:= E_ITC_MsgTypeConv.GATHERED_DATA_REQUEST,
							mLen			:= mLen);
						
		
					
ELSE
	//Unknown position send DAR with Error Report	
	GDR := GDR_Empty;
	
	// DAR
	GDR.Position	:= mpGDQ^.Position;
	GDR.eReturnCode	:= E_ErrorConv.CONFIGURATION_ERROR;

	// Reject telegram	
	M_SendData(
		meChannel := meChannelSrc,
		mMsgType  := E_ITC_MsgTypeConv.GATHERED_DATA_REQUEST,
		mpData    := ADR(GDR),
		mLen	  := mLen );
		
	// Unknown Position name received
	DebugMsg := CONCAT('GDQ - unknown Position name received: ', mpGDQ^.Position);
	fbDebugMsg.M_SendErrorMsg(mMessage := DebugMsg);
END_IF
END_METHOD

METHOD PROTECTED M_ProcessGSQ : BOOL
(**************************************************************************************
 * 	Application		:	BoxControl Framework
 *	Revision		:	$Revision: 474929 $
 *	Revision date	:	$Date: 2021-04-08 12:45:11 +0200 (tor, 08 apr 2021) $
 *	Last changed by	:	$Author: b7gessa $
 *	URL				:	$URL: http://almscdc.swisslog.com/repo/SWPD/Development/BoxControlFramework/20_Release/tags/R1.12.0/01_Software/BCF/BCF/JumpStart/20_Product/10_BCF/11_Conv/11_Com/11_ITC/FB_ITC_Conveyor.TcPOU $
 *
 *	Purpose			:	Process a received Group Status Request telegram.
 *
 * ------------------------------------------------------------------------------------
 *	Copyright Swisslog [IP AG], Switzerland. All rights reserved.
 * 
 * ------------------------------------------------------------------------------------
 *	
 * 	Revision History: 
 *
 * 	VERSION			DATE			INITIALS			DESCRIPTION
 *	0.1				01.01.2001		swl					Example
 *
 **************************************************************************************)
VAR_INPUT
	meChannelSrc		: E_MFCS_Channel; // Source communicaton channel
	mpGSQ				: POINTER TO ST_ITC_GSQ; // Pointer to GSQ
	mLen				: UDINT; // Data length
END_VAR

VAR
	meGroupNumber		: E_GroupNumber; // group number
END_VAR
// Initialize
M_ProcessGSQ := TRUE;

// Find GropuNumber of telegram
meGroupNumber := F_SearchGroupNumber(GroupName := mpGSQ^.Position);
			
// Request was for a group
// Group number valid
IF meGroupNumber > E_GroupNumber.G_BEGIN_GROUP AND 
   meGroupNumber < E_GroupNumber.G_END_GROUP THEN	
						
	// Forward to group
	M_ProcessGSQ := M_ProcessToGroup(
						meGroupNumber	:= meGroupNumber, 
						meChannelSrc	:= meChannelSrc, 
						mMsgType		:= E_ITC_MsgTypeConv.GROUP_STATUS_REQUEST,
						mpData			:= mpGSQ,
						mLen			:= mLen);
					
// Check if GCQ was sent to a SubSystem
ELSIF F_EqualSisNames(Name1 := SubsystemRegistry.SubSystemName,
                      Name2 := mpGSQ^.Position) THEN
			
	// Do for each GroupNumber
	FOR meGroupNumber := E_GroupNumber.G_BEGIN_GROUP + 1 TO E_GroupNumber.G_END_GROUP - 1 DO
		
		M_ProcessToGroup(
			meGroupNumber	:= meGroupNumber, 
			meChannelSrc	:= meChannelSrc, 
			mMsgType		:= E_ITC_MsgTypeConv.GROUP_STATUS_REQUEST,
			mpData			:= mpGSQ, 
			mLen			:= mLen);
	END_FOR
	
ELSE
	GSR := GSR_Empty;
	
	// GSR
	GSR.GroupName	:= mpGSQ^.Position;
	GSR.eReturnCode	:= E_ErrorConv.GROUPNUMBER_UNKNOWN;

	// Reject telegram	
	M_SendData(
		meChannel := meChannelSrc,
		mMsgType  := E_ITC_MsgTypeConv.GROUP_STATUS_REPORT,
		mpData    := ADR(GSR),
		mLen	  := SIZEOF(GSR));
		
	// Unknown Group name received
	DebugMsg := CONCAT('GSQ, unknown Group name received: ', mpGSQ^.Position);
	fbDebugMsg.M_SendErrorMsg(mMessage := DebugMsg);
END_IF
END_METHOD

METHOD PROTECTED M_ProcessGVQ : BOOL
(**************************************************************************************
 * 	Application		:	BoxControl Framework
 *	Revision		:	$Revision: 474929 $
 *	Revision date	:	$Date: 2021-04-08 12:45:11 +0200 (tor, 08 apr 2021) $
 *	Last changed by	:	$Author: b7gessa $
 *	URL				:	$URL: http://almscdc.swisslog.com/repo/SWPD/Development/BoxControlFramework/20_Release/tags/R1.12.0/01_Software/BCF/BCF/JumpStart/20_Product/10_BCF/11_Conv/11_Com/11_ITC/FB_ITC_Conveyor.TcPOU $
 *
 *	Purpose			:	Process a received Global Variable Request telegram.
 *
 * ------------------------------------------------------------------------------------
 *	Copyright Swisslog [IP AG], Switzerland. All rights reserved.
 * 
 * ------------------------------------------------------------------------------------
 *	
 * 	Revision History: 
 *
 * 	VERSION			DATE			INITIALS			DESCRIPTION
 *	0.1				01.01.2001		swl					Example
 *
 **************************************************************************************)
VAR_INPUT
	meChannelSrc		: E_MFCS_Channel; // Source communicaton channel
	mpGVQ				: POINTER TO ST_ITC_GVQ; // Pointer to GVQ
	mLen				: UDINT; // Data length
END_VAR

VAR
	mIdx				: INT; // Iterator
	mError				: BOOL; // Error during processing
	mVar				: ARRAY[0..9] OF DINT; // Temporary variables
END_VAR
// Initialize
M_ProcessGVQ := TRUE;

// Initialize
mError := FALSE;

// Check borders
IF mpGVQ^.Number > GVR_Table.NUMBER_OF_GVR_SIGNALS OR
   mpGVQ^.Number < 1  OR
   mpGVQ^.Quantity < 1 OR
   mpGVQ^.Quantity > 10 THEN
	// Set error
	mError := TRUE;
END_IF

// If no error is active
IF NOT mError THEN
	// If perform action is selected
	IF mpGVQ^.Code = 1 OR mpGVQ^.Code = 2 THEN
		// Map values
		mVar[0] := mpGVQ^.Variable[0];
		mVar[1] := mpGVQ^.Variable[1];
		mVar[2] := mpGVQ^.Variable[2];
		mVar[3] := mpGVQ^.Variable[3];
		mVar[4] := mpGVQ^.Variable[4];
		mVar[5] := mpGVQ^.Variable[5];
		mVar[6] := mpGVQ^.Variable[6];
		mVar[7] := mpGVQ^.Variable[7];
		mVar[8] := mpGVQ^.Variable[8];
		mVar[9] := mpGVQ^.Variable[9];
	   
		// Go trough quantity
		FOR mIdx := 0 TO mpGVQ^.Quantity - 1 DO
			// Set values
			GlobalVariable[mpGVQ^.Number, mIdx] := mVar[mIdx];
		END_FOR
	END_IF
	
	// If report state is selected
	IF mpGVQ^.Code = 0 OR mpGVQ^.Code = 2 THEN
		GVR.Number := mpGVQ^.Number;
		GVR.Quantity := mpGVQ^.Quantity;
		
		// Go trough quantity
		FOR mIdx := 0 TO 9 DO
			// Set values
			GVR.Variable[mIdx] := 0;
		END_FOR
		
		FOR mIdx := 0 TO mpGVQ^.Quantity - 1 DO
			// Set values
			GVR.Variable[mIdx] := GlobalVariable[mpGVQ^.Number, mIdx];
		END_FOR

		GVR.ReturnCode := E_ErrorConv.NO_ERROR_CODE;
	
		M_SendData(
			meChannel := meChannelSrc, 
			mMsgType  := E_ITC_MsgTypeConv.GLOBAL_VARIABLE_REPORT, 
			mpData    := ADR(GVR),
			mLen	  := SIZEOF(GVR));
	END_IF
ELSE
	GVR.Number := mpGVQ^.Number;
	GVR.Quantity := mpGVQ^.Quantity;
	GVR.Variable[0] :=0;
	GVR.Variable[1] := 0;
	GVR.Variable[2] := 0;
	GVR.Variable[3] := 0;
	GVR.Variable[4] := 0;
	GVR.Variable[5] := 0;
	GVR.Variable[6] := 0;
	GVR.Variable[7] := 0;
	GVR.Variable[8] := 0;
	GVR.Variable[9] := 0;
	GVR.ReturnCode := E_ErrorConv.WRONG_VALUE;

	M_SendData(
		meChannel := meChannelSrc, 
		mMsgType  := E_ITC_MsgTypeConv.GLOBAL_VARIABLE_REPORT, 
		mpData    := ADR(GVR),
		mLen	  := SIZEOF(GVR));
END_IF
END_METHOD

METHOD PROTECTED M_ProcessIRQ : BOOL
(**************************************************************************************
 * 	Application		:	BoxControl Framework
 *	Revision		:	$Revision: 474929 $
 *	Revision date	:	$Date: 2021-04-08 12:45:11 +0200 (tor, 08 apr 2021) $
 *	Last changed by	:	$Author: b7gessa $
 *	URL				:	$URL: http://almscdc.swisslog.com/repo/SWPD/Development/BoxControlFramework/20_Release/tags/R1.12.0/01_Software/BCF/BCF/JumpStart/20_Product/10_BCF/11_Conv/11_Com/11_ITC/FB_ITC_Conveyor.TcPOU $
 *
 *	Purpose			:	Process a received I/O Status Request telegram.
 *
 * ------------------------------------------------------------------------------------
 *	Copyright Swisslog [IP AG], Switzerland. All rights reserved.
 * 
 * ------------------------------------------------------------------------------------
 *	
 * 	Revision History: 
 *
 * 	VERSION			DATE			INITIALS			DESCRIPTION
 *	0.1				01.01.2001		swl					Example
 *
 **************************************************************************************)
VAR_INPUT
	meChannelSrc		: E_MFCS_Channel; // Source communicaton channel
	mpIRQ				: POINTER TO ST_ITC_IRQ; // Pointer to IRQ
	mLen				: UDINT; // Data length
END_VAR


VAR
	mInformation		: STRING(NUMBER_OF_ISR_DATA_LENGTH); // Internal information
	mSignalNumber		: INT; // SignalNumber
	mIdx				: INT; // Internal cunter
	mByte				: BYTE; // Internal Byte
END_VAR
// Initialize
M_ProcessIRQ := TRUE;

// Init String
mInformation := '';

// Get the signal data for each block of 4 requested
// an mDataLength of 01 actually means get 4 bits
FOR mIdx := 1 TO mpIRQ^.DataLength BY 1 DO
	
	// Calculate base signal number
	mSignalNumber  := (((mIdx - 1) * 4) + mpIRQ^.StartSignalNumber);
	// Init Byte
	mByte := 0;

	// Check if we will remain in range of the ISR Signal numbers
	IF (mSignalNumber + 4) <= NUMBER_OF_ISR_SIGNALS THEN
		// Get the signal state for this group of 4 and put them in the correct bits
		mByte.0 := ISR_SignalType[mpIRQ^.SignalType].SignalNumber[mSignalNumber];
		mByte.1 := ISR_SignalType[mpIRQ^.SignalType].SignalNumber[mSignalNumber + 1];
		mByte.2 := ISR_SignalType[mpIRQ^.SignalType].SignalNumber[mSignalNumber + 2];
		mByte.3 := ISR_SignalType[mpIRQ^.SignalType].SignalNumber[mSignalNumber + 3];
	END_IF

	// Convert the resultant tByte to a value between '0' and 'F'
	fbFormatString (sFormat := '%X', arg1 := F_BYTE(mByte));

	// Add the ASCII result for this block of 4 bits to the ISR.Information string
	mInformation := CONCAT(mInformation, fbFormatString.sOut);
END_FOR

(* Information string should always be 99 chars long
   therefore pad mInformation with trailing zeros. *)
FOR mIdx := LEN(mInformation) TO NUMBER_OF_ISR_DATA_LENGTH DO
	mInformation := CONCAT(mInformation, '0');
END_FOR

// Collect data
ISR.DataLength := mpIRQ^.DataLength;
ISR.Information := mInformation;
ISR.SignalType := mpIRQ^.SignalType;
ISR.StartSignalNumber := mpIRQ^.StartSignalNumber;
ISR.ReturnCode := E_ErrorConv.NO_ERROR_CODE;

M_SendData(
	meChannel := meChannelSrc, 
	mMsgType  := E_ITC_MsgTypeConv.I_O_STATUS_REPORT, 
	mpData    := ADR(ISR),
	mLen	  := SIZEOF(ISR));
END_METHOD

METHOD PROTECTED M_ProcessMCQ : BOOL
(**************************************************************************************
 * 	Application		:	BoxControl Framework
 *	Revision		:	$Revision: 474929 $
 *	Revision date	:	$Date: 2021-04-08 12:45:11 +0200 (tor, 08 apr 2021) $
 *	Last changed by	:	$Author: b7gessa $
 *	URL				:	$URL: http://almscdc.swisslog.com/repo/SWPD/Development/BoxControlFramework/20_Release/tags/R1.12.0/01_Software/BCF/BCF/JumpStart/20_Product/10_BCF/11_Conv/11_Com/11_ITC/FB_ITC_Conveyor.TcPOU $
 *
 *	Purpose			:	Process a received Manual Control Request telegram.
 *
 * ------------------------------------------------------------------------------------
 *	Copyright Swisslog [IP AG], Switzerland. All rights reserved.
 * 
 * ------------------------------------------------------------------------------------
 *	
 * 	Revision History: 
 *
 * 	VERSION			DATE			INITIALS			DESCRIPTION
 *	0.1				01.01.2001		swl					Example
 *
 **************************************************************************************)
VAR_INPUT
	meChannelSrc		: E_MFCS_Channel; // Source communicaton channel
	mpMCQ				: POINTER TO ST_ITC_MCQ; // Pointer to MCQ
	mLen				: UDINT; // Data length
END_VAR

VAR
	meElementNumber			: E_ElementNumber; // PositionNumber
	mFunction				: ST_PositionIdent; // Function
END_VAR

// Initialize
M_ProcessMCQ := TRUE;

// Get element number
meElementNumber := F_SearchElementPosition(ElementName := mpMCQ^.Position);

// Get function
mFunction := F_SearchFunctionPosition(Position := mpMCQ^.Position);

// Valid ElementNumber was found
IF meElementNumber > E_ElementNumber.E_BEGIN_ELEMENT AND meElementNumber < E_ElementNumber.E_END_ELEMENT THEN

	// Forward to element
	M_ProcessMCQ := M_ProcessToElement(
						meElementNumber	:= meElementNumber, 
						meChannelSrc	:= meChannelSrc, 
						mMsgType		:= E_ITC_MsgTypeConv.MANUAL_CONTROL_REQUEST,
						mpData			:= mpMCQ,
						mLen			:= mLen);		
		
// Valid FunctionNumber was found
ELSIF mFunction.eFunctionNumber > E_FunctionNumber.F_BEGIN_FUNCTION AND 
      mFunction.eFunctionNumber < E_FunctionNumber.F_END_FUNCTION THEN
	
	// Forward to function
	M_ProcessMCQ := M_ProcessToFunction(
						meFunctionNumber	:= mFunction.eFunctionNumber, 
						meChannelSrc		:= meChannelSrc, 
						mMsgType			:= E_ITC_MsgTypeConv.MANUAL_CONTROL_REQUEST,
						mpData				:= mpMCQ,
						mLen				:= mLen);
	
ELSE
	// Unknown name received
	MCR := MCR_Empty;	

	MCR.Position := mpMCQ^.Position;
	MCR.Mode := E_PositionMode.UNKNOWN_MODE;
	MCR.Code := mpMCQ^.Code;
	MCR.eReturnCode := E_ErrorConv.WRONG_VALUE;

	// Reject telegram	
	M_SendData(
		meChannel := meChannelSrc,
		mMsgType  := E_ITC_MsgTypeConv.MANUAL_CONTROL_REPORT,
		mpData    := ADR(MCR),
		mLen	  := SIZEOF(MCR));
		
	// Unknown name received
	DebugMsg := CONCAT('MCQ, unknown Position name received: ', mpMCQ^.Position);
	fbDebugMsg.M_SendErrorMsg(mMessage := DebugMsg);
END_IF
END_METHOD

METHOD PROTECTED M_ProcessRAA : BOOL
(**************************************************************************************
 * 	Application		:	BoxControl Framework
 *	Revision		:	$Revision: 474929 $
 *	Revision date	:	$Date: 2021-04-08 12:45:11 +0200 (tor, 08 apr 2021) $
 *	Last changed by	:	$Author: b7gessa $
 *	URL				:	$URL: http://almscdc.swisslog.com/repo/SWPD/Development/BoxControlFramework/20_Release/tags/R1.12.0/01_Software/BCF/BCF/JumpStart/20_Product/10_BCF/11_Conv/11_Com/11_ITC/FB_ITC_Conveyor.TcPOU $
 *
 *	Purpose			:	Process a received Transport Task Assignment telegram for a robot.
 *
 * ------------------------------------------------------------------------------------
 *	Copyright Swisslog [IP AG], Switzerland. All rights reserved.
 * 
 * ------------------------------------------------------------------------------------
 *	
 * 	Revision History: 
 *
 * VERSION DATE         INITIALS     DESCRIPTION
 * 0.0     DD.MM.YYYY   (name)       (explain customized modifications)
 *
 **************************************************************************************)

//***********************************************************************************************************
VAR_INPUT
  meChannelSrc          : E_MFCS_Channel         := 0;     // Source communicaton channel
  mpRAA                 : POINTER TO ST_ITC_RAA  := 0;     // Pointer to RAA
  mLen                  : UDINT                  := 0;     // Data length
END_VAR

//***********************************************************************************************************
VAR
  eFunctionNumber       : E_FunctionNumber       := 0;
  eElementNumber        : E_ElementNumber        := 0;
  eGroupNumber          : E_GroupNumber          := 0;
  //-------------------------------------------------------------------------------------
  Subsystem             : BOOL                   := FALSE;
END_VAR

// parse and find requested position
eFunctionNumber:= F_FindFunction  (Name:= mpRAA^.Position);
eElementNumber := F_FindElement   (Name:= mpRAA^.Position);
eGroupNumber   := F_FindGroup     (Name:= mpRAA^.Position);
Subsystem      := F_CheckSubsystem(Name:= mpRAA^.Position);

// to function ?
IF eFunctionNumber <> E_FunctionNumber.F_BEGIN_FUNCTION THEN
	M_ProcessRAA:= M_ProcessToFunction(	meFunctionNumber:= eFunctionNumber, 
										meChannelSrc    := meChannelSrc, 
										mMsgType        := E_ITC_MsgTypeConv.ROBOT_ACTION_ASSIGNMENT,
										mpData          := mpRAA, 
										mLen            := mLen);
	// forwarding successful -> no debug message necessary here


// to element ?
ELSIF eElementNumber <> E_ElementNumber.E_BEGIN_ELEMENT THEN
	M_ProcessRAA:= M_ProcessToElement(	meElementNumber:= eElementNumber,
										meChannelSrc   := meChannelSrc, 
										mMsgType       := E_ITC_MsgTypeConv.ROBOT_ACTION_ASSIGNMENT,
										mpData         := mpRAA, 
										mLen           := mLen);
	// forwarding successful -> no debug message necessary here


// to group ?
ELSIF eGroupNumber <> E_GroupNumber.G_BEGIN_GROUP THEN
	M_ProcessRAA:= M_ProcessToGroup(meGroupNumber:= eGroupNumber,
									meChannelSrc := meChannelSrc, 
									mMsgType     := E_ITC_MsgTypeConv.ROBOT_ACTION_ASSIGNMENT,
									mpData       := mpRAA, 
									mLen         := mLen);
	// forwarding successful -> no debug message necessary here


// to subsystem ?
ELSIF Subsystem THEN
	M_ProcessRAA:= M_ProcessToSubsystem(meChannelSrc:= meChannelSrc, 
										mMsgType    := E_ITC_MsgTypeConv.ROBOT_ACTION_ASSIGNMENT,
										mpData      := mpRAA, 
										mLen        := mLen);
	// forwarding successful -> no debug message necessary here


//* unknown position -> fire error telegram
ELSE
  // reject telegram
	RAC.Position        := mpRAA^.Position;
	RAC.CommandDataIndex:= mpRAA^.CommandDataIndex;
	RAC.GroupID         := mpRAA^.GroupID;
	RAC.AssignmentID    := mpRAA^.AssignmentID;
	RAC.eReturnCode     := E_ErrorConv.FUNCTIONNUMBER_UNKNOWN;
	M_SendData(	meChannel:= meChannelSrc, 
				mMsgType := E_ITC_MsgTypeConv.ROBOT_ACTION_COMPLETE, 
				mpData   := ADR(RAC),
				mLen     := SIZEOF(RAC));	

	// debug message
	// example: '11-000-0000-00-0,  unknown position addressed,  telegram = RAA,  Position = 99-999-9999-99-9,  AssignmentID = 9999999'
	DebugMsg:= '';
	DebugMsg:= CONCAT(DebugMsg, F_AddDividerToSisString(SubsystemRegistry.SubsystemName));
	DebugMsg:= CONCAT(DebugMsg, ', unknown position addressed');
	DebugMsg:= CONCAT(DebugMsg, DebugTextBlocks.TELEGRAM);
	DebugMsg:= CONCAT(DebugMsg, 'RAA');
	DebugMsg:= CONCAT(DebugMsg, DebugTextBlocks.POSITION);
	DebugMsg:= CONCAT(DebugMsg, F_AddDividerToSisString(Name:= mpRAA^.Position)  );
	DebugMsg:= CONCAT(DebugMsg, DebugTextBlocks.ASSIGNMENTID);
	DebugMsg:= CONCAT(DebugMsg, UDINT_TO_STRING(mpRAA^.AssignmentID) );
	fbDebugMsg.M_SendErrorMsg(mMessage := DebugMsg);
	
	// forwarding to here ITC were possible so prevent error message from FB_SIS_MsgManager
	M_ProcessRAA:= TRUE;
END_IF
END_METHOD

METHOD PROTECTED M_ProcessRDQ : BOOL
(**************************************************************************************
 * 	Application		:	BoxControl Framework
 *	Revision		:	$Revision: 474929 $
 *	Revision date	:	$Date: 2021-04-08 12:45:11 +0200 (tor, 08 apr 2021) $
 *	Last changed by	:	$Author: b7gessa $
 *	URL				:	$URL: http://almscdc.swisslog.com/repo/SWPD/Development/BoxControlFramework/20_Release/tags/R1.12.0/01_Software/BCF/BCF/JumpStart/20_Product/10_BCF/11_Conv/11_Com/11_ITC/FB_ITC_Conveyor.TcPOU $
 *
 *	Purpose			:	Robot delete request
 *
 * ------------------------------------------------------------------------------------
 *	Copyright Swisslog [IP AG], Switzerland. All rights reserved.
 * 
 * ------------------------------------------------------------------------------------
 *	
 * 	Revision History: 
 *
 * 	VERSION			DATE			INITIALS			DESCRIPTION
 *	0.1				03.11.2015		Kay Röder			Example
 *
 **************************************************************************************)
VAR_INPUT
	meChannelSrc				: E_MFCS_Channel; // Source communicaton channel
	mpRDQ						: POINTER TO ST_ITC_RDQ; // Pointer to EDQ
	mLen						: UDINT; // Data length
END_VAR

VAR
	mMsgPosition		: ST_PositionIdent; // Function position
	mReturnCode 		: U_ErrorCode;
END_VAR
// Initialize
M_ProcessRDQ := TRUE;
	   
// Get position from message
mMsgPosition := F_SearchFunctionPosition(Position := mpRDQ^.Position);
	
// If a valid function was found with a valid zone
IF 	mMsgPosition.eFunctionNumber > E_FunctionNumber.F_BEGIN_FUNCTION AND 
	mMsgPosition.eFunctionNumber < E_FunctionNumber.F_END_FUNCTION AND 
	mMsgPosition.ZoneNumber >= 0 AND mMsgPosition.ZoneNumber <= NUMBER_OF_ZONES_PER_FUNCTION THEN
	
	// Forward to element
	M_ProcessRDQ := M_ProcessToFunction(
						meFunctionNumber	:= mMsgPosition.eFunctionNumber, 
						meChannelSrc		:= meChannelSrc, 
						mMsgType			:= E_ITC_MsgTypeConv.ROBOT_DELETE_REQUEST,
						mpData				:= mpRDQ, 
						mLen				:= mLen);
				
	DebugMsg := CONCAT('Robot Delete Assignment Request: ', UDINT_TO_STRING(mpRDQ^.AssignmentID));
	fbDebugMsg.M_SendInfoMsg(mMessage := DebugMsg);
 
ELSE
	mReturnCode.Conv := E_ErrorConv.FUNCTIONNUMBER_UNKNOWN; 
	
	// Reject telegram	
	RDR.Position := mpRDQ^.Position;
	RDR.CommandDataIndex := mpRDQ^.CommandDataIndex;
	RDR.GroupID := mpRDQ^.GroupID;
	RDR.AssignmentID := 0;
	RDR.ReturnCode := mReturnCode.Conv;

	M_SendData(
		meChannel := meChannelSrc, 
		mMsgType  := E_ITC_MsgTypeConv.ROBOT_DELETE_REPORT, 
		mpData    := ADR(RDR),
		mLen	  := SIZEOF(RDR));

	DebugMsg := CONCAT('Robot Delete Assignment Request: ', UDINT_TO_STRING(mpRDQ^.AssignmentID));
	DebugMsg := CONCAT(DebugMsg, 'has an invalid ITC config on RowPaQ-PLC-project');
	fbDebugMsg.M_SendErrorMsg(mMessage := DebugMsg);
END_IF
END_METHOD

METHOD PROTECTED M_ProcessSCQ : BOOL
(**************************************************************************************
 * 	Application		:	BoxControl Framework
 *	Revision		:	$Revision: 474929 $
 *	Revision date	:	$Date: 2021-04-08 12:45:11 +0200 (tor, 08 apr 2021) $
 *	Last changed by	:	$Author: b7gessa $
 *	URL				:	$URL: http://almscdc.swisslog.com/repo/SWPD/Development/BoxControlFramework/20_Release/tags/R1.12.0/01_Software/BCF/BCF/JumpStart/20_Product/10_BCF/11_Conv/11_Com/11_ITC/FB_ITC_Conveyor.TcPOU $
 *
 *	Purpose			:	Process a received Subsystem Control Request telegram.
 *
 * ------------------------------------------------------------------------------------
 *	Copyright Swisslog [IP AG], Switzerland. All rights reserved.
 * 
 * ------------------------------------------------------------------------------------
 *	
 * 	Revision History: 
 *
 * 	VERSION			DATE			INITIALS			DESCRIPTION
 *	0.1				01.01.2001		swl					Example
 *
 **************************************************************************************)
VAR_INPUT
	meChannelSrc		: E_MFCS_Channel; // Source communicaton channel
	mpSCQ				: POINTER TO ST_ITC_SCQ; // Pointer to SCQ
	mLen				: UDINT; // Data length
END_VAR
// Initialize 
M_ProcessSCQ := TRUE;

// Check if SubSystem is valid
IF F_EqualSisNames(Name1 := SubsystemRegistry.SubSystemName,
                   Name2 := mpSCQ^.SubsystemName) THEN
		
	// Forward to subsystem
	M_ProcessSCQ := M_ProcessToSubsystem(
						meChannelSrc	:= meChannelSrc, 
						mMsgType		:= E_ITC_MsgTypeConv.SUBSYSTEM_CONTROL_REQUEST,
						mpData			:= mpSCQ,
						mLen			:= mLen);		
ELSE
	// Unknown SubSystem number received
	SCR.SubsystemName	:= mpSCQ^.SubsystemName;
	SCR.Code			:= mpSCQ^.Code;
	SCR.Variable		:= mpSCQ^.Variable;
	SCR.ReturnCode		:= E_ErrorConv.SubsystemNUMBER_UNKNOWN;

	// Reject telegram	
	M_SendData(
		meChannel := meChannelSrc,
		mMsgType  := E_ITC_MsgTypeConv.SUBSYSTEM_CONTROL_REPLY,
		mpData    := ADR(SCR),
		mLen	  := SIZEOF(SCR));

	// Unknown SubSystem number received
	DebugMsg := CONCAT('SCQ, unknown SubSystem name received: ', mpSCQ^.SubsystemName);
	fbDebugMsg.M_SendErrorMsg(mMessage := DebugMsg);
END_IF
END_METHOD

METHOD PROTECTED M_ProcessSDO : BOOL
(**************************************************************************************
 * 	Application		:	BoxControl Framework
 *	Revision		:	$Revision: 474929 $
 *	Revision date	:	$Date: 2021-04-08 12:45:11 +0200 (tor, 08 apr 2021) $
 *	Last changed by	:	$Author: b7gessa $
 *	URL				:	$URL: http://almscdc.swisslog.com/repo/SWPD/Development/BoxControlFramework/20_Release/tags/R1.12.0/01_Software/BCF/BCF/JumpStart/20_Product/10_BCF/11_Conv/11_Com/11_ITC/FB_ITC_Conveyor.TcPOU $
 *
 *	Purpose			:	Process a received Set Digital Output telegram.
 *						Set or Reset the appropriate SDO signal number according 
 *						to the data in the telegram
 *
 * ------------------------------------------------------------------------------------
 *	Copyright Swisslog [IP AG], Switzerland. All rights reserved.
 * 
 * ------------------------------------------------------------------------------------
 *	
 * 	Revision History: 
 *
 * 	VERSION			DATE			INITIALS			DESCRIPTION
 *	0.1				01.01.2001		swl					Example
 *
 **************************************************************************************)
VAR_INPUT
	meChannelSrc		: E_MFCS_Channel; // Source communicaton channel
	mpSDO				: POINTER TO ST_ITC_SDO; // Pointer to SCQ
	mLen				: UDINT; // Data length
END_VAR
// Initialize
M_ProcessSDO := TRUE;

// Range check the SignalNumber
IF mpSDO^.SignalNumber > 0 THEN
	// Set SignalState
	SDOSignalNumber[mpSDO^.SignalNumber] := INT_TO_BOOL(mpSDO^.SignalState);
END_IF
END_METHOD

METHOD PROTECTED M_ProcessSIQ : BOOL
(**************************************************************************************
 * 	Application		:	BoxControl Framework
 *	Revision		:	$Revision: 474929 $
 *	Revision date	:	$Date: 2021-04-08 12:45:11 +0200 (tor, 08 apr 2021) $
 *	Last changed by	:	$Author: b7gessa $
 *	URL				:	$URL: http://almscdc.swisslog.com/repo/SWPD/Development/BoxControlFramework/20_Release/tags/R1.12.0/01_Software/BCF/BCF/JumpStart/20_Product/10_BCF/11_Conv/11_Com/11_ITC/FB_ITC_Conveyor.TcPOU $
 *
 *	Purpose			:	Process a received Scanner Information Request telegram.
 *
 * ------------------------------------------------------------------------------------
 *	Copyright Swisslog [IP AG], Switzerland. All rights reserved.
 * 
 * ------------------------------------------------------------------------------------
 *	
 * 	Revision History: 
 *
 * 	VERSION			DATE			INITIALS			DESCRIPTION
 *	0.1				01.01.2001		swl					Example
 *
 **************************************************************************************)
VAR_INPUT
	meChannelSrc		: E_MFCS_Channel; // Source communicaton channel
	mpSIQ				: POINTER TO ST_ITC_SIQ; // Pointer to SIQ
	mLen				: UDINT; // Data length
END_VAR

VAR
	mFunction			: ST_PositionIdent; // Function position
END_VAR
// Initialize
M_ProcessSIQ := TRUE;

//Find element function of telegram
mFunction := F_SearchFunctionPosition(Position := mpSIQ^.Position);

// If function number is valid
IF mFunction.eFunctionNumber > E_FunctionNumber.F_BEGIN_FUNCTION AND 
   mFunction.eFunctionNumber < E_FunctionNumber.F_END_FUNCTION THEN
   
	// Forward to function
	M_ProcessSIQ := M_ProcessToFunction(
						meFunctionNumber	:= mFunction.eFunctionNumber,
						meChannelSrc		:= meChannelSrc, 
						mMsgType			:= E_ITC_MsgTypeConv.SCANNER_INFORMATION_REQUEST,
						mpData				:= mpSIQ, 
						mLen				:= mLen);

ELSE
	// Unknown Position name received
	SIR.Position := mpSIQ^.Position;
	SIR.Code := mpSIQ^.Code;
	SIR.TU_ID := '';
	SIR.Counter1 := 0;
	SIR.Counter2 := 0;
	SIR.Counter3 := 0;
	SIR.Counter4 := 0;
	SIR.Counter5 := 0;
	SIR.eReturnCode := E_ErrorConv.FUNCTIONNUMBER_UNKNOWN;

	// Reject telegram	
	M_SendData(
		meChannel := meChannelSrc,
		mMsgType  := E_ITC_MsgTypeConv.SCANNER_INFORMATION_REPORT,
		mpData    := ADR(SIR),
		mLen	  := SIZEOF(SIR));

	// Unknown Position name received
	DebugMsg := CONCAT('SIQ, unknown Position name received: ', mpSIQ^.Position);
	fbDebugMsg.M_SendErrorMsg(mMessage := DebugMsg);	
END_IF
END_METHOD

METHOD PROTECTED M_ProcessSSQ : BOOL
(**************************************************************************************
 * 	Application		:	BoxControl Framework
 *	Revision		:	$Revision: 474929 $
 *	Revision date	:	$Date: 2021-04-08 12:45:11 +0200 (tor, 08 apr 2021) $
 *	Last changed by	:	$Author: b7gessa $
 *	URL				:	$URL: http://almscdc.swisslog.com/repo/SWPD/Development/BoxControlFramework/20_Release/tags/R1.12.0/01_Software/BCF/BCF/JumpStart/20_Product/10_BCF/11_Conv/11_Com/11_ITC/FB_ITC_Conveyor.TcPOU $
 *
 *	Purpose			:	Process a received Subsystem Status Request telegram.
 *
 * ------------------------------------------------------------------------------------
 *	Copyright Swisslog [IP AG], Switzerland. All rights reserved.
 * 
 * ------------------------------------------------------------------------------------
 *	
 * 	Revision History: 
 *
 * 	VERSION			DATE			INITIALS			DESCRIPTION
 *	0.1				01.01.2001		swl					Example
 *
 **************************************************************************************)
VAR_INPUT
	meChannelSrc		: E_MFCS_Channel; // Source communicaton channel
	mpSSQ				: POINTER TO ST_ITC_SSQ; // Pointer to SCQ
	mLen				: UDINT; // Data length
END_VAR
// Initialize
M_ProcessSSQ := TRUE;

// Check if SubSystem is valid
IF F_EqualSisNames(Name1 := SubsystemRegistry.SubsystemName,
                   Name2 := mpSSQ^.Position) THEN
		
		// Forward to subsystem
		M_ProcessSSQ := M_ProcessToSubsystem(
							meChannelSrc	:= meChannelSrc, 
							mMsgType		:= E_ITC_MsgTypeConv.SUBSYSTEM_STATUS_REQUEST,
							mpData			:= mpSSQ, 
							mLen			:= mLen);	
ELSE
	SSR := SSR_Empty;
	
	// SSR
	SSR.SubsystemName	:= mpSSQ^.Position;
	SSR.eReturnCode	:= E_ErrorConv.SubsystemNUMBER_UNKNOWN;

	// Reject telegram	
	M_SendData(
		meChannel := meChannelSrc,
		mMsgType  := E_ITC_MsgTypeConv.SUBSYSTEM_STATUS_REPORT,
		mpData    := ADR(SSR),
		mLen	  := SIZEOF(SSR));
		
	// Unknown SubSystem number received
	DebugMsg := CONCAT('SSQ, unknown SubSystem name received: ', mpSSQ^.Position);
	fbDebugMsg.M_SendErrorMsg(mMessage := DebugMsg);
END_IF
END_METHOD

METHOD PROTECTED M_ProcessTDQ : BOOL
(**************************************************************************************
 *  Application     :   BoxControl Framework
 *  Revision date   :   $Date: 2021-04-08 12:45:11 +0200 (tor, 08 apr 2021) $
 *  Author          :   CDC
 * ------------------------------------------------------------------------------------
 *  © Swisslog AG
 *  Swisslog is not liable for any usage of this source code that is not agreed 
 *  on between Swisslog and the other party. The mandatory legal liability remains 
 *  unaffected.
 * ------------------------------------------------------------------------------------
 *  Revision History: 
 *
 *  VERSION DATE         INITIALS     DESCRIPTION
 *  0.0     DD.MM.YYYY   (name)       (explain customized modifications)
 *
 **************************************************************************************)
VAR_INPUT
	meChannelSrc			: E_MFCS_Channel; // Source communicaton channel
	mpTDQ					: POINTER TO ST_ITC_TDQ; // Pointer to TDQ
	mLen					: UDINT; // Data length
END_VAR

VAR
	mPosition				: ST_PositionIdent ; // Position
	mReturnCode				: E_ErrorConv; // Return code
	mTU_ID_Present			: BOOL; // TU-ID present
	mTU_DataIndex			: DINT; // TU-data index
	mAssignmentID_Present	: BOOL; // Assignment-ID present
	mAssignmentID_Index		: DINT; // Assignment-ID index
END_VAR
// Init
mReturnCode := E_ErrorConv.NO_ERROR_CODE;
M_ProcessTDQ := TRUE;
mTU_ID_Present := FALSE;
mTU_DataIndex := 0;
mAssignmentID_Present := FALSE;
mAssignmentID_Index := 0;

// Get position from telegram
mPosition := F_SearchFunctionPosition( Position := mpTDQ^.Position);

// Order to delete all TU-data
IF mpTDQ^.Code = 1 THEN
	// Check no function number and unknown TU-ID
	IF mpTDQ^.TU_ID = Conveyor.TU_ID_UNKNOWN AND mPosition.eFunctionNumber = 0 THEN
		// Check all TU-Data for DataSets
		FOR mTU_DataIndex := 1 TO Conveyor.NUMBER_OF_TU_DATA BY 1 DO
			// Check if TU-DataSet is used
			IF TU_DataTable[mTU_DataIndex].DataSet.DataPresent THEN	
				// debug message: '11-001-0095-01-1,  TU_DataIndex deleted,  telegram = TDQ,  TU_DataIndex = 5,  TuID = 000012345,  AssignmentID = 999999999'
				DebugMsg := '';
				DebugMsg := CONCAT(DebugMsg, F_AddDividerToSisString(mpTDQ^.Position));
				DebugMsg := CONCAT(DebugMsg, ',  TU_DataIndex deleted');
				DebugMsg := CONCAT(DebugMsg, DebugTextBlocks.TELEGRAM);
				DebugMsg := CONCAT(DebugMsg, 'TDQ');
				DebugMsg := CONCAT(DebugMsg, F_CreateTU_DataString(TU_DataIndex:= mTU_DataIndex));
				fbDebugMsg.M_SendInfoMsg(DebugMsg);
				// Delete TU-Data
				F_DeleteTU_Data(
					TU_DataIndex 	:= mTU_DataIndex, // TU_DataIndex from zone
					NoTTC 			:= FALSE); // No TTC will be sent
			END_IF
		END_FOR

		TDR.Position := mpTDQ^.Position;
		TDR.TU_ID := mpTDQ^.TU_ID;
		TDR.AssignmentID := mpTDQ^.AssignmentID;
		TDR.MsgSequence := mpTDQ^.MsgSequence;
		TDR.ReturnCode := mReturnCode;
		
		M_SendData(
			meChannel := meChannelSrc, 
			mMsgType  := E_ITC_MsgTypeConv.TASK_DELETE_REPORT, 
			mpData    := ADR(TDR),
			mLen	  := SIZEOF(TDR));
		RETURN;
	ELSE
		// Error: Wrong value
		mReturnCode := E_ErrorConv.WRONG_VALUE;
	END_IF
	
// Specific request for TU-ID or position
ELSE
	// Check if an Assignment-ID is present
	mAssignmentID_Present := mpTDQ^.AssignmentID > 0 AND mpTDQ^.AssignmentID < Conveyor.ASSIGNMENT_ID_UNKNOWN;
	
	// Check if a TU-ID is present
	mTU_ID_Present := mpTDQ^.TU_ID <> F_StuffString('', Conveyor.TU_ID_STRINGLENGTH,'0', FALSE) AND
				      mpTDQ^.TU_ID <> F_StuffString('', Conveyor.TU_ID_STRINGLENGTH,' ', FALSE);
	
	// If a valid position is found
	IF mPosition.eFunctionNumber > E_FunctionNumber.F_BEGIN_FUNCTION AND
	   mPosition.ZoneNumber > 0 THEN
		// Get TU-data from zone
		mTU_DataIndex := F_GetTU_DataIndex(
								eFunctionNumber := mPosition.eFunctionNumber, // PositionNumber
								ZoneNumber := mPosition.ZoneNumber); // ZoneNumber
		// A TU index was found
		IF mTU_DataIndex > 0 THEN
			IF mAssignmentID_Present THEN
				// Compare received Assignment ID with the Assignment ID from the position
				IF TU_DataTable[mTU_DataIndex].AssignmentID <> mpTDQ^.AssignmentID THEN
					// Error: Wrong Assignement-ID
					mReturnCode := E_ErrorConv.ASSIGNMENT_ID_WRONG;
				END_IF
			ELSIF mTU_ID_Present THEN
				// Compare received TU ID with the TU ID from the position
				IF TU_DataTable[mTU_DataIndex].TU_ID.ASCII <> mpTDQ^.TU_ID THEN
					// Error: Wrong TU-ID
					mReturnCode := E_ErrorConv.TU_ID_WRONG;
				END_IF
			ELSE
				// Error: Wrong value
				mReturnCode := E_ErrorConv.ID_WRONG;
			END_IF
		ELSE
			// Error: No TU data set available on position
			mReturnCode := E_ErrorConv.EMPTY_TU_DATA_SET;
		END_IF
		
	// Request to subsystem
	ELSIF mpTDQ^.Position <> F_ReduceToAlphaNumeric(SubsystemRegistry.SubsystemName) THEN
		// Error: Position wrong 
		mReturnCode := E_ErrorConv.FUNCTIONNUMBER_UNKNOWN;
		
	// Telegram without function number
	ELSE
		IF mAssignmentID_Present THEN
			// Search TU-data index based on the Assignement-ID in the TU-data table
			mAssignmentID_Index := F_SearchAssignmentId(mpTDQ^.AssignmentID);
		END_IF
		
		IF mTU_ID_Present THEN
			// Search TU-data index based on the TU-ID in the TU-data table
			mTU_DataIndex := F_SearchTU_ByHashCode(mpTDQ^.TU_ID);
		END_IF			
		
		// If an Assignement-ID index is found
		IF mAssignmentID_Index <> 0 THEN
			// Search position belonging to the Assignement-ID index
			// to report last position
			mPosition := F_SearchPositionOfTU_Index(
								TU_DataIndex := mAssignmentID_Index, // TU_DataIndex from zone
								eStartFunctionNumber := E_FunctionNumber.F_BEGIN_FUNCTION + 1); // Start Zone
		// If a TU-data index is found
		ELSIF mTU_DataIndex <> 0 THEN
			// Search position belonging to the TU-data index
			// to report last position
			mPosition := F_SearchPositionOfTU_Index(
								TU_DataIndex := mTU_DataIndex, // TU_DataIndex from zone
								eStartFunctionNumber := E_FunctionNumber.F_BEGIN_FUNCTION + 1); // Start Zone
		ELSE
			IF mAssignmentID_Present THEN
				// Error: Wrong Assignement-ID
				mReturnCode := E_ErrorConv.ASSIGNMENT_ID_WRONG;
			ELSIF mTU_ID_Present THEN
				// Error: Wrong TU-ID
				mReturnCode := E_ErrorConv.TU_ID_WRONG;
			ELSE
				// Error: No data
				mReturnCode := E_ErrorConv.ID_WRONG;
			END_IF
		END_IF
	END_IF
END_IF

// Send task delete report
IF mPosition.eFunctionNumber <> E_FunctionNumber.F_BEGIN_FUNCTION THEN
	TDR.Position := F_ReduceToAlphaNumeric(FunctionRegistry[mPosition.eFunctionNumber].Zone[mPosition.ZoneNumber].ZoneName);
ELSE
	TDR.Position := mpTDQ^.Position;
END_IF
TDR.TU_ID := mpTDQ^.TU_ID;
TDR.AssignmentID := mpTDQ^.AssignmentID;
TDR.MsgSequence := mpTDQ^.MsgSequence;
TDR.ReturnCode := mReturnCode;

M_SendData(
	meChannel := meChannelSrc, 
	mMsgType  := E_ITC_MsgTypeConv.TASK_DELETE_REPORT, 
	mpData    := ADR(TDR),
	mLen	  := SIZEOF(TDR));

// Still no error so far
IF mReturnCode = 0  THEN
	// TU-data index available
	IF mTU_DataIndex <> 0 THEN
		// debug message: '11-001-0095-01-1,  TU_DataIndex deleted,  telegram = TDQ,  TU_DataIndex = 5,  TuID = 000012345,  AssignmentID = 999999999'
		DebugMsg := '';
		DebugMsg := CONCAT(DebugMsg, F_AddDividerToSisString(mpTDQ^.Position));
		DebugMsg := CONCAT(DebugMsg, ',  TU_DataIndex deleted');
		DebugMsg := CONCAT(DebugMsg, DebugTextBlocks.TELEGRAM);
		DebugMsg := CONCAT(DebugMsg, 'TDQ');
		DebugMsg := CONCAT(DebugMsg, F_CreateTU_DataString(TU_DataIndex:= mTU_DataIndex));
		fbDebugMsg.M_SendInfoMsg(DebugMsg);
		// Delete TU-data in the system
		F_DeleteTU_Data(
			TU_DataIndex 	:= mTU_DataIndex,
			NoTTC 			:= FALSE);
	// Assignement-ID index available
	ELSIF mAssignmentID_Index <> 0 THEN
		// debug message: '11-001-0095-01-1,  TU_DataIndex deleted,  telegram = TDQ,  TU_DataIndex = 5,  TuID = 000012345,  AssignmentID = 999999999'
		DebugMsg := '';
		DebugMsg := CONCAT(DebugMsg, F_AddDividerToSisString(mpTDQ^.Position));
		DebugMsg := CONCAT(DebugMsg, ',  TU_DataIndex deleted');
		DebugMsg := CONCAT(DebugMsg, DebugTextBlocks.TELEGRAM);
		DebugMsg := CONCAT(DebugMsg, 'TDQ');
		DebugMsg := CONCAT(DebugMsg, F_CreateTU_DataString(TU_DataIndex:= mAssignmentID_Index));
		fbDebugMsg.M_SendInfoMsg(DebugMsg);
		// Delete TU-data in the system
		F_DeleteTU_Data(
			TU_DataIndex 	:= mAssignmentID_Index,
			NoTTC 			:= FALSE);
	ELSE		
		DebugMsg := 'TDQ, Process failed - no TU-index available.';
		fbDebugMsg.M_SendErrorMsg(mMessage := DebugMsg);		
	END_IF
END_IF
END_METHOD

METHOD PROTECTED M_ProcessToElement : BOOL
(**************************************************************************************
 * 	Application		:	BoxControl Framework
 *	Revision		:	$Revision: 474929 $
 *	Revision date	:	$Date: 2021-04-08 12:45:11 +0200 (tor, 08 apr 2021) $
 *	Last changed by	:	$Author: b7gessa $
 *	URL				:	$URL: http://almscdc.swisslog.com/repo/SWPD/Development/BoxControlFramework/20_Release/tags/R1.12.0/01_Software/BCF/BCF/JumpStart/20_Product/10_BCF/11_Conv/11_Com/11_ITC/FB_ITC_Conveyor.TcPOU $
 *
 *	Purpose			:	ITC - Process message to element
 *
 * ------------------------------------------------------------------------------------
 *	Copyright Swisslog [IP AG], Switzerland. All rights reserved.
 * 
 * ------------------------------------------------------------------------------------
 *	
 * 	Revision History: 
 *
 * 	VERSION			DATE			INITIALS			DESCRIPTION
 *	0.1				01.01.2001		swl					Example
 *
 **************************************************************************************)
VAR_INPUT
	meElementNumber	: E_ElementNumber;
	meChannelSrc	: E_MFCS_Channel; // Source communicaton channel
	mMsgType			: INT; // msg type
	mpData				: POINTER TO PVOID; // data pointer
	mLen				: UDINT; // Data length
END_VAR

VAR
	mrefObject		: REFERENCE TO FB_BaseObject; // Reference
END_VAR
// Initialize
M_ProcessToElement := TRUE;

// Check if ElementNumber is valid
IF meElementNumber > E_ElementNumber.E_BEGIN_ELEMENT AND 
   meElementNumber < E_ElementNumber.E_END_ELEMENT THEN
	// Set reference
	mrefObject REF= ElementRegistry[meElementNumber].rElement;
	
	// Check if reference is valid
	IF __ISVALIDREF(mrefObject) THEN
			// Forward message to corresponding object
		M_ProcessToElement := mrefObject.M_ITC_ProcessMsg(
								meChannelSrc := meChannelSrc,
								mMsgType	 := mMsgType,
								mpData		 := mpData,
								mLen		 := mLen); 
	END_IF	
END_IF
END_METHOD

METHOD PROTECTED M_ProcessToFunction : BOOL
(**************************************************************************************
 * 	Application		:	BoxControl Framework
 *	Revision		:	$Revision: 474929 $
 *	Revision date	:	$Date: 2021-04-08 12:45:11 +0200 (tor, 08 apr 2021) $
 *	Last changed by	:	$Author: b7gessa $
 *	URL				:	$URL: http://almscdc.swisslog.com/repo/SWPD/Development/BoxControlFramework/20_Release/tags/R1.12.0/01_Software/BCF/BCF/JumpStart/20_Product/10_BCF/11_Conv/11_Com/11_ITC/FB_ITC_Conveyor.TcPOU $
 *
 *	Purpose			:	ITC - Process message to function
 *
 * ------------------------------------------------------------------------------------
 *	Copyright Swisslog [IP AG], Switzerland. All rights reserved.
 * 
 * ------------------------------------------------------------------------------------
 *	
 * 	Revision History: 
 *
 * 	VERSION			DATE			INITIALS			DESCRIPTION
 *	0.1				01.01.2001		swl					Example
 *
 **************************************************************************************)
VAR_INPUT
	meFunctionNumber	: E_FunctionNumber; // Function number
	meChannelSrc		: E_MFCS_Channel; // Source communicaton channel
	mMsgType			: INT; // msg type
	mpData				: POINTER TO PVOID; // data pointer
	mLen				: UDINT; // Data length
END_VAR

VAR
	mrefObject			: REFERENCE TO FB_BaseObject; // Reference
END_VAR
// Initialize
M_ProcessToFunction := TRUE;

// If a valid function was found with a valid zone
IF 	meFunctionNumber > E_FunctionNumber.F_BEGIN_FUNCTION AND 
	meFunctionNumber < E_FunctionNumber.F_END_FUNCTION THEN

	// Set reference 
	mrefObject REF= FunctionRegistry[meFunctionNumber].rFunction;
	
	// Check if reference is valid
	IF __ISVALIDREF(mrefObject) THEN

		// Call M_ITC_AddToBuffer
		M_ProcessToFunction := mrefObject.M_ITC_ProcessMsg(
								meChannelSrc := meChannelSrc, // Number of the source 
								mMsgType	 := mMsgType, // Type of the ITC message
								mpData		 := mpData,
								mLen		 := mLen); // Data pointer of the message	
	END_IF
END_IF
END_METHOD

METHOD PROTECTED M_ProcessToGroup : BOOL
(**************************************************************************************
 * 	Application		:	BoxControl Framework
 *	Revision		:	$Revision: 474929 $
 *	Revision date	:	$Date: 2021-04-08 12:45:11 +0200 (tor, 08 apr 2021) $
 *	Last changed by	:	$Author: b7gessa $
 *	URL				:	$URL: http://almscdc.swisslog.com/repo/SWPD/Development/BoxControlFramework/20_Release/tags/R1.12.0/01_Software/BCF/BCF/JumpStart/20_Product/10_BCF/11_Conv/11_Com/11_ITC/FB_ITC_Conveyor.TcPOU $
 *
 *	Purpose			:	ITC - Process message to group
 *
 * ------------------------------------------------------------------------------------
 *	Copyright Swisslog [IP AG], Switzerland. All rights reserved.
 * 
 * ------------------------------------------------------------------------------------
 *	
 * 	Revision History: 
 *
 * 	VERSION			DATE			INITIALS			DESCRIPTION
 *	0.1				01.01.2001		swl					Example
 *
 **************************************************************************************)
VAR_INPUT
	meGroupNumber		: E_GroupNumber; // Groupnumber
	meChannelSrc		: E_MFCS_Channel; // Source communicaton channel
	mMsgType			: INT; // msg type
	mpData				: POINTER TO PVOID; // data pointer
	mLen				: UDINT; // Data length
END_VAR

VAR
	mrefObject			: REFERENCE TO FB_BaseObject; // Reference
END_VAR
// Initialize
M_ProcessToGroup := TRUE;

// Check if GroupNumber is valid
IF meGroupNumber > E_GroupNumber.G_BEGIN_GROUP AND 
   meGroupNumber < E_GroupNumber.G_END_GROUP THEN
	// Set reference
	mrefObject REF= GroupRegistry[meGroupNumber].rGroup;
	
	// Check if reference is valid
	IF __ISVALIDREF(mrefObject) THEN
		
		// Send ITC-message to a specified group
		M_ProcessToGroup := mrefObject.M_ITC_ProcessMsg(
								meChannelSrc := meChannelSrc,
								mMsgType	 := mMsgType, 
								mpData		 := mpData,
								mLen		 := mLen); 
	END_IF
END_IF
END_METHOD

METHOD PROTECTED M_ProcessToSubsystem : BOOL
(**************************************************************************************
 * 	Application		:	BoxControl Framework
 *	Revision		:	$Revision: 474929 $
 *	Revision date	:	$Date: 2021-04-08 12:45:11 +0200 (tor, 08 apr 2021) $
 *	Last changed by	:	$Author: b7gessa $
 *	URL				:	$URL: http://almscdc.swisslog.com/repo/SWPD/Development/BoxControlFramework/20_Release/tags/R1.12.0/01_Software/BCF/BCF/JumpStart/20_Product/10_BCF/11_Conv/11_Com/11_ITC/FB_ITC_Conveyor.TcPOU $
 *
 *	Purpose			:	ITC - Process message to subsystem
 *
 * ------------------------------------------------------------------------------------
 *	Copyright Swisslog [IP AG], Switzerland. All rights reserved.
 * 
 * ------------------------------------------------------------------------------------
 *	
 * 	Revision History: 
 *
 * 	VERSION			DATE			INITIALS			DESCRIPTION
 *	0.1				01.01.2001		swl					Example
 *
 **************************************************************************************)
VAR_INPUT
	meChannelSrc		: E_MFCS_Channel; // Source communicaton channel
	mMsgType			: INT; // msg type
	mpData				: POINTER TO PVOID; // data pointer
	mLen				: UDINT; // Data length
END_VAR

VAR
	mrefObject			: REFERENCE TO FB_BaseObject; // Reference
END_VAR
// Initialize
M_ProcessToSubsystem := TRUE;

// Set reference 
mrefObject REF= SubsystemRegistry.rSubsystem;

// Check if reference is valid
IF __ISVALIDREF(mrefObject) THEN
	// Call M_ITC_AddToBuffer
	M_ProcessToSubsystem := mrefObject.M_ITC_ProcessMsg(
								meChannelSrc := meChannelSrc,
								mMsgType	 := mMsgType, 
								mpData		 := mpData,	
								mLen		 := mLen);  
END_IF
END_METHOD

METHOD PROTECTED M_ProcessTTA : BOOL
(**************************************************************************************
 * 	Application		:	BoxControl Framework
 *	Revision		:	$Revision: 474929 $
 *	Revision date	:	$Date: 2021-04-08 12:45:11 +0200 (tor, 08 apr 2021) $
 *	Last changed by	:	$Author: b7gessa $
 *	URL				:	$URL: http://almscdc.swisslog.com/repo/SWPD/Development/BoxControlFramework/20_Release/tags/R1.12.0/01_Software/BCF/BCF/JumpStart/20_Product/10_BCF/11_Conv/11_Com/11_ITC/FB_ITC_Conveyor.TcPOU $
 *
 *	Purpose			:	Process a received Transport Task Assignment telegram.
 *
 * ------------------------------------------------------------------------------------
 *	Copyright Swisslog [IP AG], Switzerland. All rights reserved.
 * 
 * ------------------------------------------------------------------------------------
 *	
 * 	Revision History: 
 *
 * VERSION DATE         INITIALS     DESCRIPTION
 * 0.0     DD.MM.YYYY   (name)       (explain customized modifications)
 *
 **************************************************************************************)
VAR_INPUT
	meChannelSrc				: E_MFCS_Channel; // Source communicaton channel
	mpTTA						: POINTER TO ST_ITC_TTA; // Pointer to TTA
	mLen						: UDINT;
END_VAR

VAR
	mOtherPosition				: ST_PositionIdent; // OtherPosition where same Index is used
	mDestinationPosition		: ARRAY[1..NUMBER_OF_DESTINATIONS] OF ST_PositionIdent; // DestinationPosition
	mVirtualDestinationPosition	: ARRAY[1..NUMBER_OF_DESTINATIONS] OF ST_PositionIdent;
	mReturnCode					: E_ErrorConv; // Error code
	mTU_DataIndexPosition		: DINT; // Data Index from PositionNumber
	mTU_DataIndex				: DINT; // Data Index from Data_ID
	mRequestForPosition			: BOOL; // Request for a Position
	mTransportData				: ST_TransportControlData; // Transport data
	mTU_ID_Present				: BOOL; // TU-ID present
	mAssignmentID_Present		: BOOL; // Assignment ID present
	mAssignmentID_Index			: DINT; // Assignment ID index
	mDestIndex					: INT; // Temporary destination index
END_VAR
// Initialize
M_ProcessTTA := TRUE;
mTU_DataIndexPosition := 0;
mRequestForPosition := FALSE;	
mTU_DataIndex := 0;
mAssignmentID_Index := 0;
mAssignmentID_Present := FALSE;
mTU_ID_Present := FALSE;

(**************************************************************************************
Check if request is valid
***************************************************************************************)
// Search position in registry
Position := F_SearchFunctionPosition(Position := mpTTA^.Position);

//Check if a TU-ID is present
mTU_ID_Present := 	mpTTA^.TU_ID <> F_StuffString('', Conveyor.TU_ID_STRINGLENGTH,'0', FALSE)
				AND mpTTA^.TU_ID <> F_StuffString('', Conveyor.TU_ID_STRINGLENGTH,' ', FALSE);

IF mTU_ID_Present THEN
	// Search if the TU-ID already exists
	mTU_DataIndex := F_SearchTU_ByHashCode(mpTTA^.TU_ID);
END_IF	

// Check if an asssignment-ID is present					   
mAssignmentID_Present := mpTTA^.AssignmentID > 0;

IF mAssignmentID_Present THEN
	// Search if the assignment-ID already exists
	mAssignmentID_Index := F_SearchAssignmentId(mpTTA^.AssignmentID);
END_IF


// If the telegram contains no TU-ID and no assignment-ID
IF NOT mTU_ID_Present AND NOT mAssignmentID_Present THEN
	// Error: ID is wrong 
	mReturnCode := E_ErrorConv.ID_WRONG;
	// debug message: '11-000-0000-00-0,  TuID and AssignmentID missing,  telegram = TTA'
	DebugMsg:= '';
	DebugMsg:= CONCAT(DebugMsg, F_AddDividerToSisString(SubsystemRegistry.SubsystemName));
	DebugMsg:= CONCAT(DebugMsg, ',  TuID and AssignmentID missing');
	DebugMsg:= CONCAT(DebugMsg, DebugTextBlocks.TELEGRAM);
	DebugMsg:= CONCAT(DebugMsg, 'TTA');
	fbDebugMsg.M_SendErrorMsg(mMessage := DebugMsg);


// If the request goes to a position
ELSIF Position.eFunctionNumber > E_FunctionNumber.F_BEGIN_FUNCTION AND 
	Position.eFunctionNumber < E_FunctionNumber.F_END_FUNCTION THEN
	// If a valid zone was found
	IF 	Position.ZoneNumber > 0
	AND Position.ZoneNumber <= NUMBER_OF_ZONES_PER_FUNCTION THEN
		// Get transport data
		mTransportData := F_GetTransportControlData(
		eFunctionNumber := Position.eFunctionNumber,
		ZoneNumber		:= Position.ZoneNumber);
		
		(*	Data can only be added if the location is physically occupied.
			State occupied is not working in this place, because on a system
			with enabled MFC, the place gets occupied only with a physical 
			and a logical unit. *)
		IF mTransportData.SensorOccupied THEN
			// Save - Valid request for a position
			mRequestForPosition := TRUE;	

			// Get TU Index of telegram position
			mTU_DataIndexPosition := F_GetTU_DataIndex( 
			eFunctionNumber := Position.eFunctionNumber,
			ZoneNumber 		:= Position.ZoneNumber);
			// If an index is found
			IF mTU_DataIndexPosition > 0 THEN
			(* 
			Adding data is allowed, if
			- TU-ID of desired position is 'unknown' OR
			- Telegram TU-ID is equal to position TU-ID
			
			AND
			- Position consists of an unknown assignment-ID OR
			- Assignment-ID is equal to the requested one		
			
			AND
			- When a requested Index was available, it needs to be equal to position index		
			*)
				IF (TU_DataTable[mTU_DataIndexPosition].TU_ID.ASCII = Conveyor.TU_ID_UNKNOWN OR 
				mpTTA^.TU_ID = TU_DataTable[mTU_DataIndexPosition].TU_ID.ASCII) AND 
				(mpTTA^.AssignmentID = TU_DataTable[mTU_DataIndexPosition].AssignmentID OR
				Conveyor.ASSIGNMENT_ID_UNKNOWN = TU_DataTable[mTU_DataIndexPosition].AssignmentID) AND
				((mpTTA^.TU_DataIndex > 0 AND mpTTA^.TU_DataIndex = mTU_DataIndexPosition) OR (mpTTA^.TU_DataIndex = 0)) THEN 
					// Adding data is allowed by TU-ID
					;
				// Adding not allowed
				ELSE
					// When the assignment-ID was not equal to the already existing or 
					// the assignment-ID on the position was not unknown
					IF TU_DataTable[mTU_DataIndexPosition].AssignmentID <> mpTTA^.AssignmentID AND 
					   TU_DataTable[mTU_DataIndexPosition].AssignmentID <> Conveyor.ASSIGNMENT_ID_UNKNOWN THEN
						// Error: Assignment-ID is false 
						mReturnCode := E_ErrorConv.ASSIGNMENT_ID_WRONG;
						// debug message: '11-001-0120-01-0,  AssignmentID mismatch,  telegram = TTA,  expected = 112233,  current = 332211'
						DebugMsg:= '';
						DebugMsg:= CONCAT(DebugMsg, F_AddDividerToSisString(Position.PositionName));
						DebugMsg:= CONCAT(DebugMsg, ',  AssignmentID mismatch');
						DebugMsg:= CONCAT(DebugMsg, DebugTextBlocks.TELEGRAM);
						DebugMsg:= CONCAT(DebugMsg, 'TTA');
						DebugMsg:= CONCAT(DebugMsg, DebugTextBlocks.EXPECTED);
						DebugMsg:= CONCAT(DebugMsg, UDINT_TO_STRING(TU_DataTable[mTU_DataIndexPosition].AssignmentID) );
						DebugMsg:= CONCAT(DebugMsg, DebugTextBlocks.CURRENT);
						DebugMsg:= CONCAT(DebugMsg, UDINT_TO_STRING(mpTTA^.AssignmentID) );
						fbDebugMsg.M_SendErrorMsg(mMessage := DebugMsg);

					// Otherwise its because of a wrong TU-ID
					// - Not equal
					// - Not unknown
					ELSIF TU_DataTable[mTU_DataIndexPosition].TU_ID.ASCII <> Conveyor.TU_ID_UNKNOWN AND 
						  TU_DataTable[mTU_DataIndexPosition].TU_ID.ASCII <> mpTTA^.TU_ID THEN
						// Error: TU-ID is false 
						mReturnCode := E_ErrorConv.TU_ID_WRONG;
						// debug message: '11-001-0120-01-0,  TuID mismatch,  telegram = TTA,  expected = 112233,  current = 332211'
						DebugMsg:= '';
						DebugMsg:= CONCAT(DebugMsg, F_AddDividerToSisString(Position.PositionName));
						DebugMsg:= CONCAT(DebugMsg, ',  TuID mismatch');
						DebugMsg:= CONCAT(DebugMsg, DebugTextBlocks.TELEGRAM);
						DebugMsg:= CONCAT(DebugMsg, 'TTA');
						DebugMsg:= CONCAT(DebugMsg, DebugTextBlocks.EXPECTED);
						DebugMsg:= CONCAT(DebugMsg, TU_DataTable[mTU_DataIndexPosition].TU_ID.ASCII);
						DebugMsg:= CONCAT(DebugMsg, DebugTextBlocks.CURRENT);
						DebugMsg:= CONCAT(DebugMsg, mpTTA^.TU_ID);
						fbDebugMsg.M_SendErrorMsg(mMessage := DebugMsg);

					// Otherwise, requested index was wrong
					ELSE
						mReturnCode := E_ErrorConv.WRONG_VALUE;
						// debug message: '11-001-0120-01-0,  TU_DataIndex mismatch,  telegram = TTA,  expected = 1,  current = 3'
						DebugMsg:= '';
						DebugMsg:= CONCAT(DebugMsg, F_AddDividerToSisString(Position.PositionName));
						DebugMsg:= CONCAT(DebugMsg, ',  TU_DataIndex mismatch');
						DebugMsg:= CONCAT(DebugMsg, DebugTextBlocks.TELEGRAM);
						DebugMsg:= CONCAT(DebugMsg, 'TTA');
						DebugMsg:= CONCAT(DebugMsg, DebugTextBlocks.EXPECTED);
						DebugMsg:= CONCAT(DebugMsg, DINT_TO_STRING(mTU_DataIndexPosition)  );
						DebugMsg:= CONCAT(DebugMsg, DebugTextBlocks.CURRENT);
						DebugMsg:= CONCAT(DebugMsg, DINT_TO_STRING(mpTTA^.TU_DataIndex)  );
						fbDebugMsg.M_SendErrorMsg(mMessage := DebugMsg);
					END_IF		
				END_IF
			END_IF 
		ELSE
			// Error: Zone free
			mReturnCode := E_ErrorConv.POSITION_NOT_CORRECT_OCCUPIED;
			// debug message: '11-001-0120-01-0,  position is not occupied,  telegram = TTA'
			DebugMsg:= '';
			DebugMsg:= CONCAT(DebugMsg, F_AddDividerToSisString(Position.PositionName));
			DebugMsg:= CONCAT(DebugMsg, ',  position is not occupied');
			DebugMsg:= CONCAT(DebugMsg, DebugTextBlocks.TELEGRAM);
			DebugMsg:= CONCAT(DebugMsg, 'TTA');
			fbDebugMsg.M_SendErrorMsg(mMessage := DebugMsg);
		END_IF

	ELSE
		// Error: Position wrong 
		mReturnCode := E_ErrorConv.FUNCTIONNUMBER_UNKNOWN;
		// debug message: '11-000-0000-00-0,  unknown position addressed,  telegram = TTA,  Position = 99-999-9999-99-9'
		DebugMsg:= '';
		DebugMsg:= CONCAT(DebugMsg, F_AddDividerToSisString(SubsystemRegistry.SubsystemName));
		DebugMsg:= CONCAT(DebugMsg, ',  unknown position addressed');
		DebugMsg:= CONCAT(DebugMsg, DebugTextBlocks.TELEGRAM);
		DebugMsg:= CONCAT(DebugMsg, 'TTA');
		DebugMsg:= CONCAT(DebugMsg, DebugTextBlocks.POSITION);
		DebugMsg:= CONCAT(DebugMsg, F_AddDividerToSisString(Name:= mpTTA^.Position)  );
		fbDebugMsg.M_SendErrorMsg(mMessage := DebugMsg);
	END_IF

// If the request goes to the subsystem MM-000-0000-00-0
ELSIF NOT F_EqualSisNames(Name1:= mpTTA^.Position,
						  Name2:= SubsystemRegistry.SubsystemName) THEN
	// Error: Position wrong 
	mReturnCode := E_ErrorConv.FUNCTIONNUMBER_UNKNOWN; 
	// debug message: '00-000-0000-00-0,  unknown position addressed,  telegram = TTA,  Position = 99-999-9999-99-9'
	DebugMsg:= '';
	DebugMsg:= CONCAT(DebugMsg, '00-000-0000-00-0');  // subsystem is not properly addressed
	DebugMsg:= CONCAT(DebugMsg, ',  unknown position addressed');
	DebugMsg:= CONCAT(DebugMsg, DebugTextBlocks.TELEGRAM);
	DebugMsg:= CONCAT(DebugMsg, 'TTA');
	DebugMsg:= CONCAT(DebugMsg, DebugTextBlocks.POSITION);
	DebugMsg:= CONCAT(DebugMsg, F_AddDividerToSisString(Name:= mpTTA^.Position)  );
	fbDebugMsg.M_SendErrorMsg(mMessage := DebugMsg);

// TU-data index update request to subsystem
ELSIF mpTTA^.TU_DataIndex > 0 THEN
	// Validate corresponding index
	IF TU_DataTable[mpTTA^.TU_DataIndex].DataSet.DataPresent THEN
		(* If the received telegram contains two existing IDs (Assignment and TU) -> both have to match to the same index. *)
		IF mTU_DataIndex > 0 AND mAssignmentID_Index > 0 THEN
			IF mTU_DataIndex <> mAssignmentID_Index THEN
				mReturnCode := E_ErrorConv.WRONG_VALUE;	
				// debug message: '11-000-0000-00-0,  AssignmentID mismatch,  telegram = TTA,  expected = 87654321,  current = 12345678'
				DebugMsg:= '';
				DebugMsg:= CONCAT(DebugMsg, F_AddDividerToSisString(SubsystemRegistry.SubsystemName));
				DebugMsg:= CONCAT(DebugMsg, ',  AssignmentID mismatch');
				DebugMsg:= CONCAT(DebugMsg, DebugTextBlocks.TELEGRAM);
				DebugMsg:= CONCAT(DebugMsg, 'TTA');
				DebugMsg:= CONCAT(DebugMsg, DebugTextBlocks.EXPECTED);
				DebugMsg:= CONCAT(DebugMsg, UDINT_TO_STRING(TU_DataTable[mTU_DataIndex].AssignmentID)  );
				DebugMsg:= CONCAT(DebugMsg, DebugTextBlocks.CURRENT);
				DebugMsg:= CONCAT(DebugMsg, UDINT_TO_STRING(mpTTA^.AssignmentID)  );
				fbDebugMsg.M_SendErrorMsg(mMessage := DebugMsg);

			// Compare found index to TTA index
			ELSIF mpTTA^.TU_DataIndex <> mTU_DataIndex THEN
				mReturnCode := E_ErrorConv.WRONG_VALUE;	
				// debug message: '11-000-0000-00-0,  TU_DataIndex mismatch,  telegram = TTA,  expected = 1,  current = 3'
				DebugMsg:= '';
				DebugMsg:= CONCAT(DebugMsg, F_AddDividerToSisString(SubsystemRegistry.SubsystemName));
				DebugMsg:= CONCAT(DebugMsg, ',  TU_DataIndex mismatch');
				DebugMsg:= CONCAT(DebugMsg, DebugTextBlocks.TELEGRAM);
				DebugMsg:= CONCAT(DebugMsg, 'TTA');
				DebugMsg:= CONCAT(DebugMsg, DebugTextBlocks.EXPECTED);
				DebugMsg:= CONCAT(DebugMsg, DINT_TO_STRING(mTU_DataIndex)  );
				DebugMsg:= CONCAT(DebugMsg, DebugTextBlocks.CURRENT);
				DebugMsg:= CONCAT(DebugMsg, DINT_TO_STRING(mpTTA^.TU_DataIndex)  );
				fbDebugMsg.M_SendErrorMsg(mMessage := DebugMsg);
			END_IF

		// When an TU-ID index was found
		ELSIF mTU_DataIndex > 0 THEN
			// Compare found index to TTA index
			IF mTU_DataIndex <> mpTTA^.TU_DataIndex THEN
				mReturnCode := E_ErrorConv.WRONG_VALUE;	
				// debug message: '11-000-0000-00-0,  TU_DataIndex mismatch,  telegram = TTA,  expected = 1,  current = 3'
				DebugMsg:= '';
				DebugMsg:= CONCAT(DebugMsg, F_AddDividerToSisString(SubsystemRegistry.SubsystemName));
				DebugMsg:= CONCAT(DebugMsg, ',  TU_DataIndex mismatch');
				DebugMsg:= CONCAT(DebugMsg, DebugTextBlocks.TELEGRAM);
				DebugMsg:= CONCAT(DebugMsg, 'TTA');
				DebugMsg:= CONCAT(DebugMsg, DebugTextBlocks.EXPECTED);
				DebugMsg:= CONCAT(DebugMsg, DINT_TO_STRING(mTU_DataIndex)  );
				DebugMsg:= CONCAT(DebugMsg, DebugTextBlocks.CURRENT);
				DebugMsg:= CONCAT(DebugMsg, DINT_TO_STRING(mpTTA^.TU_DataIndex)  );
				fbDebugMsg.M_SendErrorMsg(mMessage := DebugMsg);
			END_IF

		// When an assignment-ID index was found
		ELSIF mAssignmentID_Index > 0 THEN
			// Compare found index to TTA index
			IF mAssignmentID_Index <> mpTTA^.TU_DataIndex THEN
				mReturnCode := E_ErrorConv.WRONG_VALUE;	
				// debug message: '11-000-0000-00-0,  AssignmentID mismatch,  telegram = TTA,  expected = 87654321,  current = 12345678'
				DebugMsg:= '';
				DebugMsg:= CONCAT(DebugMsg, F_AddDividerToSisString(SubsystemRegistry.SubsystemName));
				DebugMsg:= CONCAT(DebugMsg, ',  AssignmentID mismatch');
				DebugMsg:= CONCAT(DebugMsg, DebugTextBlocks.TELEGRAM);
				DebugMsg:= CONCAT(DebugMsg, 'TTA');
				DebugMsg:= CONCAT(DebugMsg, DebugTextBlocks.EXPECTED);
				DebugMsg:= CONCAT(DebugMsg, UDINT_TO_STRING(TU_DataTable[mAssignmentID_Index].AssignmentID)  );
				DebugMsg:= CONCAT(DebugMsg, DebugTextBlocks.CURRENT);
				DebugMsg:= CONCAT(DebugMsg, UDINT_TO_STRING(mpTTA^.AssignmentID)  );
				fbDebugMsg.M_SendErrorMsg(mMessage := DebugMsg);
			END_IF
		END_IF

		IF mReturnCode = 0 THEN
			// Validate TU-ID
			IF (TU_DataTable[mpTTA^.TU_DataIndex].TU_ID.ASCII <> Conveyor.TU_ID_UNKNOWN AND mpTTA^.TU_ID <> TU_DataTable[mpTTA^.TU_DataIndex].TU_ID.ASCII)
			 OR(TU_DataTable[mpTTA^.TU_DataIndex].AssignmentID <> Conveyor.ASSIGNMENT_ID_UNKNOWN AND mpTTA^.AssignmentID <> TU_DataTable[mpTTA^.TU_DataIndex].AssignmentID) THEN
				IF (TU_DataTable[mpTTA^.TU_DataIndex].TU_ID.ASCII <> Conveyor.TU_ID_UNKNOWN AND
				mpTTA^.TU_ID <> TU_DataTable[mpTTA^.TU_DataIndex].TU_ID.ASCII) THEN
					// Error: TU-ID is false 
					mReturnCode := E_ErrorConv.TU_ID_WRONG;
					// debug message: '11-001-0120-01-0,  TuID mismatch,  telegram = TTA,  expected = 112233,  current = 332211'
					DebugMsg:= '';
					DebugMsg:= CONCAT(DebugMsg, F_AddDividerToSisString(SubsystemRegistry.SubsystemName));
					DebugMsg:= CONCAT(DebugMsg, ',  TuID mismatch');
					DebugMsg:= CONCAT(DebugMsg, DebugTextBlocks.TELEGRAM);
					DebugMsg:= CONCAT(DebugMsg, 'TTA');
					DebugMsg:= CONCAT(DebugMsg, DebugTextBlocks.EXPECTED);
					DebugMsg:= CONCAT(DebugMsg, TU_DataTable[mpTTA^.TU_DataIndex].TU_ID.ASCII);
					DebugMsg:= CONCAT(DebugMsg, DebugTextBlocks.CURRENT);
					DebugMsg:= CONCAT(DebugMsg, mpTTA^.TU_ID);
					fbDebugMsg.M_SendErrorMsg(mMessage := DebugMsg);

